(* IEC 61131-3 sources: Mizera_Tube/Plc (part 6) *)

(* ---- usrLoad.plc ---- *)
#funcdec "FLP.plc"
#funcdec "SPist.plc"

#include "usrMem.inc"
#include "Iol.inc"

VAR_IN_OUT
#include "usrIol.inc"
#include "mem.inc"
END_VAR

VAR
M1_M2_M3_MOVE:        SINGLE_PISTON;
CenteringPist1:       SINGLE_PISTON;
CenteringPist2:       SINGLE_PISTON;
CenteringPist3:       SINGLE_PISTON;
CenteringPist4:       SINGLE_PISTON;
Sup_G_Pist:           SINGLE_PISTON;
Pist_F_FB:            SINGLE_PISTON;
J_VEL_SWITCH:                    FF;
TON_CHAIN:                      TON;
TON_INVERTER_FIL:               TON;
TON_INVERTER_FIL1:              TON;
END_VAR

FUNCTION LOADER
************************************************************
* Loader Initialization Selection
************************************************************
PAGE_PLC

************************************************************
* Loader arms to be back (Arms J)
************************************************************
LD     ch0_ValFunM
EQ     330
OR(
LD     ch8_ValFunM
EQ     330
)
OR(
LD     ch0_ValFunM                * Arms J Going Back Slow
EQ     431
)
OR(
LD     ch0_ValFunM                * whole loader homming
EQ     445
)
AND    PRGRUN_CN0
ANDN   PRGSTOP_CN0
OR(
LD     BtnGuiM1M2M3_Open
ANDN   PRGRUN_CN0
)
ANDN   I_I_M1_M2_M3_OPEN
ST     O_O_M1_M2_M3_Open

LDN    I_I_M1_M2_M3_OPEN
AND(
LD     %ax30.ra92
LT     SUPPORT_4_Quota
)
ANDN   %cn0.rc8.0
ANDN   ch0_in_ref
S      %PLCmsg8.5

************************************************************
* Loader arms to be in machine (Arms J)
************************************************************
LD     ch0_ValFunM
EQ     331
OR(
LD     ch8_ValFunM
EQ     331
)
AND    PRGRUN_CN0
ANDN   PRGSTOP_CN0
OR(
LD     BtnGuiM1M2M3_Close
ANDN   PRGRUN_CN0
)
ANDN   I_I_M1_M2_M3_CLOSE
ST     O_O_M1_M2_M3_Close

CAL    TON_INVERTER_FIL(IN=I_I_M1_M2_M3_ALARM, PT=300)
LD     TON_INVERTER_FIL.Q
S      %PLCerr21.8

************************************************************
* Loader arms speed control
************************************************************
LD     O_O_M1_M2_M3_Close
OR(
       LD     ch0_ValFunM
       EQ     431                 * Slow Chain Backward
       AND    O_O_M1_M2_M3_Open
)
ANDN(
       LD     ch0_ValFunM
       EQ     330
       OR(
       LD     ch8_ValFunM
       EQ     330
       )
	   OR(
       LD     ch0_ValFunM                * whole loader homming
       EQ     445
       )
)
ORN    %cn0.rc8.0
ST     O_O_Arm_Slow

LDN    O_O_Arm_Slow
ST     O_O_Arm_Fast

************************************************************
* Loader chain to be inside (D)
************************************************************
LD     ch0_ValFunM
EQ     443
OR(
LD     ch8_ValFunM
EQ     443
)
AND    PRGRUN_CN0
ANDN   PRGSTOP_CN0
OR(
LD     BtnGuiChainForw
ANDN   I_I_TubeOnChain_D
ANDN   PRGRUN_CN0
)
ST     O_O_Chain_Forw_D

CAL    TON_CHAIN(IN=O_O_Chain_Forw_D,PT=20000) *20S
LD     TON_CHAIN.Q
AND    PRGRUN_CN0
S      STORE_Empty

CAL    TON_INVERTER_FIL1(IN=I_I_Loader_Alarm, PT=300)
LD     TON_INVERTER_FIL1.Q
S      %PLCerr21.9

************************************************************
* Loader chain to be outside (D)
************************************************************
LD     ch0_ValFunM
EQ     444
OR(
LD     ch8_ValFunM
EQ     444
)
AND    PRGRUN_CN0
ANDN   PRGSTOP_CN0
ANDN   I_I_HomeChain_E
OR(
LD     BtnGuiChainBackw
ANDN   PRGRUN_CN0
)
ST     O_O_Chain_Back_D

************************************************************
* Centering Piston 1
************************************************************
LD     PRGRUN_CN0                     ** M0.0 cn0.rc8.0  Programma in corso
ST     CenteringPist1.xAuto

LD     Pul_Reset                      ** (gPlc0.3)Reset pushbutton
OR     Pul_Start                      ** (gPlc0.1)Start pushbutton
ST     CenteringPist1.xReset

LD     BtnGuiCentering_Open_1
OR     BtnGuiCentering_Open_All
OR     Force_Open_Center_1
ST     CenteringPist1.xManualPlus

LD     BtnGuiCentering_Close_1
OR     BtnGuiCentering_Cls_All
ANDN   Force_Open_Center_1
ST     CenteringPist1.xManualMinus

LD     Fun_M332_Ch0
OR(
LD     ch8_ValFunM
EQ     332
)
OR     Fun_M445_Ch0
OR     Force_Open_Center_1
OR     Fun_M452_Ch0                   ** Open all centering
ST     CenteringPist1.xAutoPlus

LD     Fun_M333_Ch0
OR(
LD     ch8_ValFunM
EQ     333
)
OR     Fun_M455_Ch0
ST     CenteringPist1.xAutoMinus

LD     I_I_PRESSIONE_ARIA_IMPIANTO    ** **(Common for all pistons) %USR_M0
ST     CenteringPist1.xAirPressure

LD     I_I_Centering_Open_1
ST     CenteringPist1.xSensorPlus

LD     %PLCFLAGS.1
ST     CenteringPist1.xSensorMinus

LD     %PLCFLAGS.1
ST     CenteringPist1.xPlusAtInit

LD     %PLCFLAGS.1
ST     CenteringPist1.xSingleEffect

LD     10000
ST     CenteringPist1.xTimeOut

LDN    I_I_EMERGENZA                  ** Machine OK (no EMERG.)
ST     CenteringPist1.xEmerg

CAL    CenteringPist1

LD     CenteringPist1.yPistonPlus
ST     O_O_Centering_Open_1

LD     CenteringPist1.yPistonMinus
ST     O_O_Centering_Close_1

LD     CenteringPist1.yAlarm
ST     %PLCerr21.10

************************************************************
* Centering Piston 2
************************************************************
LD     PRGRUN_CN0                     ** M0.0 cn0.rc8.0  Programma in corso
ST     CenteringPist2.xAuto

LD     Pul_Reset                      ** (gPlc0.3)Reset pushbutton
OR     Pul_Start                      ** (gPlc0.1)Start pushbutton
ST     CenteringPist2.xReset

LD     BtnGuiCentering_Open_2
OR     BtnGuiCentering_Open_All
OR     Force_Open_Center_2
ST     CenteringPist2.xManualPlus

LD     BtnGuiCentering_Close_2
OR     BtnGuiCentering_Cls_All
ANDN   Force_Open_Center_2
ST     CenteringPist2.xManualMinus

LD     Fun_M446_Ch0
OR(
LD     ch8_ValFunM
EQ     446
)
OR     Fun_M445_Ch0
OR     Force_Open_Center_2
OR     Fun_M452_Ch0                   ** Open all centering
ST     CenteringPist2.xAutoPlus

LD     Fun_M447_Ch0
OR(
LD     ch8_ValFunM
EQ     447
)
OR     Fun_M455_Ch0
ST     CenteringPist2.xAutoMinus

LD     I_I_PRESSIONE_ARIA_IMPIANTO    ** **(Common for all pistons) %USR_M0
ST     CenteringPist2.xAirPressure

LD     I_I_Centering_Open_2
ST     CenteringPist2.xSensorPlus

LD     %PLCFLAGS.1
ST     CenteringPist2.xSensorMinus

LD     %PLCFLAGS.1
ST     CenteringPist2.xPlusAtInit

LD     %PLCFLAGS.1
ST     CenteringPist2.xSingleEffect

LD     10000
ST     CenteringPist2.xTimeOut

LDN    I_I_EMERGENZA                  ** Machine OK (no EMERG.)
ST     CenteringPist2.xEmerg

CAL    CenteringPist2

LD     CenteringPist2.yPistonPlus
ST     O_O_Centering_Open_2

LD     CenteringPist2.yPistonMinus
ST     O_O_Centering_Close_2

LD     CenteringPist2.yAlarm
ST     %PLCerr21.11

************************************************************
* Centering Piston 3
************************************************************
LD     PRGRUN_CN0                     ** M0.0 cn0.rc8.0  Programma in corso
ST     CenteringPist3.xAuto

LD     Pul_Reset                      ** (gPlc0.3)Reset pushbutton
OR     Pul_Start                      ** (gPlc0.1)Start pushbutton
ST     CenteringPist3.xReset

LD     BtnGuiCentering_Open_3
OR     BtnGuiCentering_Open_All
OR     Force_Open_Center_3
ST     CenteringPist3.xManualPlus

LD     BtnGuiCentering_Close_3
OR     BtnGuiCentering_Cls_All
ANDN   Force_Open_Center_3
ST     CenteringPist3.xManualMinus

LD     Fun_M448_Ch0
OR(
LD     ch8_ValFunM
EQ     448
)
OR     Fun_M445_Ch0
OR     Force_Open_Center_3
OR     Fun_M452_Ch0                   ** Open all centering
ST     CenteringPist3.xAutoPlus

LD     Fun_M449_Ch0
OR(
LD     ch8_ValFunM
EQ     449
)
OR     Fun_M455_Ch0
ST     CenteringPist3.xAutoMinus

LD     I_I_PRESSIONE_ARIA_IMPIANTO    ** **(Common for all pistons) %USR_M0
ST     CenteringPist3.xAirPressure

LD     I_I_Centering_Open_3
ST     CenteringPist3.xSensorPlus

LD     %PLCFLAGS.1
ST     CenteringPist3.xSensorMinus

LD     %PLCFLAGS.1
ST     CenteringPist3.xPlusAtInit

LD     %PLCFLAGS.1
ST     CenteringPist3.xSingleEffect

LD     10000
ST     CenteringPist3.xTimeOut

LDN    I_I_EMERGENZA                  ** Machine OK (no EMERG.)
ST     CenteringPist3.xEmerg

CAL    CenteringPist3

LD     CenteringPist3.yPistonPlus
ST     O_O_Centering_Open_3

LD     CenteringPist3.yPistonMinus
ST     O_O_Centering_Close_3

LD     CenteringPist3.yAlarm
ST     %PLCerr21.12

************************************************************
* Centering Piston 4
************************************************************
LD     PRGRUN_CN0                     ** M0.0 cn0.rc8.0  Programma in corso
ST     CenteringPist4.xAuto

LD     Pul_Reset                      ** (gPlc0.3)Reset pushbutton
OR     Pul_Start                      ** (gPlc0.1)Start pushbutton
ST     CenteringPist4.xReset

LD     BtnGuiCentering_Open_4
OR     BtnGuiCentering_Open_All
OR     Force_Open_Center_4
ST     CenteringPist4.xManualPlus

LD     BtnGuiCentering_Close_4
OR     BtnGuiCentering_Cls_All
ANDN   Force_Open_Center_4
ST     CenteringPist4.xManualMinus

LD     Fun_M450_Ch0
OR(
LD     ch8_ValFunM
EQ     450
)
OR     Fun_M445_Ch0
OR     Force_Open_Center_4
OR     Fun_M452_Ch0                   ** Open all centering
ST     CenteringPist4.xAutoPlus

LD     Fun_M451_Ch0
OR(
LD     ch8_ValFunM
EQ     451
)
OR     Fun_M455_Ch0
ST     CenteringPist4.xAutoMinus

LD     I_I_PRESSIONE_ARIA_IMPIANTO    ** **(Common for all pistons) %USR_M0
ST     CenteringPist4.xAirPressure

LD     I_I_Centering_Open_4
ST     CenteringPist4.xSensorPlus

LD     %PLCFLAGS.1
ST     CenteringPist4.xSensorMinus

LD     %PLCFLAGS.1
ST     CenteringPist4.xPlusAtInit

LD     %PLCFLAGS.1
ST     CenteringPist4.xSingleEffect

LD     10000
ST     CenteringPist4.xTimeOut

LDN    I_I_EMERGENZA                  ** Machine OK (no EMERG.)
ST     CenteringPist4.xEmerg

CAL    CenteringPist4

LD     CenteringPist4.yPistonPlus
ST     O_O_Centering_Open_4

LD     CenteringPist4.yPistonMinus
ST     O_O_Centering_Close_4

LD     CenteringPist4.yAlarm
ST     %PLCerr21.13

************************************************************
* Support ( G up / down )
************************************************************
LD     PRGRUN_CN0                     ** M0.0 cn0.rc8.0  Programma in corso
ST     Sup_G_Pist.xAuto

LD     Pul_Reset                      ** (gPlc0.3)Reset pushbutton
OR     Pul_Start                      ** (gPlc0.1)Start pushbutton
ST     Sup_G_Pist.xReset

LD     BtnGui_G_Up
ST     Sup_G_Pist.xManualPlus

LD     BtnGui_G_Dwn
ST     Sup_G_Pist.xManualMinus

LD     Fun_M334_Ch0
OR(
LD     ch8_ValFunM
EQ     334
)
ST     Sup_G_Pist.xAutoPlus          * Up

LD     Fun_M335_Ch0
OR(
LD     ch8_ValFunM
EQ     335
)
OR     Fun_M445_Ch0
ST     Sup_G_Pist.xAutoMinus         * Dwn

LD     I_I_PRESSIONE_ARIA_IMPIANTO    ** **(Common for all pistons) %USR_M0
ST     Sup_G_Pist.xAirPressure

LD     I_I_CylinderUp_G
ST     Sup_G_Pist.xSensorPlus

LD     I_I_CylinderDwn_G
ST     Sup_G_Pist.xSensorMinus

LD     %PLCFLAGS.0
ST     Sup_G_Pist.xPlusAtInit

LD     %PLCFLAGS.1
ST     Sup_G_Pist.xSingleEffect

LD     10000
ST     Sup_G_Pist.xTimeOut

LDN    I_I_EMERGENZA                  ** Machine OK (no EMERG.)
ST     Sup_G_Pist.xEmerg

CAL    Sup_G_Pist

LD     Sup_G_Pist.yPistonPlus
*ANDN   I_I_CylinderUp_G
ST     O_O_CylinderUp_G

LD     Sup_G_Pist.yPistonMinus
*ANDN   I_I_CylinderDwn_G
ST     O_O_CylinderDwn_G

LD     Sup_G_Pist.yAlarm
ST     %PLCerr20.13

************************************************************
* Support F (Forward/Backward)
************************************************************
LD     PRGRUN_CN0                     ** M0.0 cn0.rc8.0  Programma in corso
ST     Pist_F_FB.xAuto

LD     Pul_Reset                      ** (gPlc0.3)Reset pushbutton
OR     Pul_Start                      ** (gPlc0.1)Start pushbutton
ST     Pist_F_FB.xReset

LD     BtnGui_F_Forw
ST     Pist_F_FB.xManualPlus

LD     BtnGui_F_Backw
ST     Pist_F_FB.xManualMinus

LD     Fun_M434_Ch0
OR(
LD     ch8_ValFunM
EQ     434
)
ST     Pist_F_FB.xAutoPlus

LD     Fun_M435_Ch0
OR(
LD     ch8_ValFunM
EQ     435
)
OR(
LD     ch0_ValFunM                    * whole loader homming
EQ     445
)
ST     Pist_F_FB.xAutoMinus

LD     I_I_PRESSIONE_ARIA_IMPIANTO    ** **(Common for all pistons) %USR_M0
ST     Pist_F_FB.xAirPressure

LD     I_I_CylinderForw_F
ST     Pist_F_FB.xSensorPlus

LD     I_I_CylinderBack_F
ST     Pist_F_FB.xSensorMinus

LD     %PLCFLAGS.1
ST     Pist_F_FB.xPlusAtInit

LD     %PLCFLAGS.1
ST     Pist_F_FB.xSingleEffect

LD     10000
ST     Pist_F_FB.xTimeOut

LDN    I_I_EMERGENZA                  ** Machine OK (no EMERG.)
ST     Pist_F_FB.xEmerg

CAL    Pist_F_FB

LD     Pist_F_FB.yPistonPlus
ANDN   I_I_CylinderForw_F
ST     O_O_CylinderForw_F

LD     Pist_F_FB.yPistonMinus
ANDN   I_I_CylinderBack_F
ST     O_O_CylinderBack_F

LD     Pist_F_FB.yAlarm
ST     %PLCerr20.14

************************************************************
* Alarm / Status Reset
************************************************************
LD     Pul_Reset
ST     O_O_Rst_InverterAlm
R      %PLCmsg8.5
R      %PLCerr21.8
R      %PLCerr21.9
R      ISO_Loader_Retrace
R      iso_G510_Running
R      iso_G520_V_Unload
R      iso_G580_Running

LD     Pul_Reset
ORN    PRGRUN_CN0
R      STORE_Empty
R      TubeOnGworklist

LD     BtnClrLoaderBreakPoint
ANDN   %cn0.rc8.0
JMPCN  CLRLDSTATUS
LD     0
ST     LoaderProcess
CLRLDSTATUS:

END_FUNCTION

(* ---- usrMdec.plc ---- *)
**************************************************
********* READ M FROM ISO ************************
**************************************************
#defcom %rc9 Register M function
#defcom %rc8.4 Strobe M function

#include "usrMem.inc"

VAR_IN_OUT
#include "mem.inc"
END_VAR

VAR
Register_M_Ch0	             AT %cn0.rc9;
Strobe_M_Ch0  	             AT %cn0.rc8.4;
Register_M_Ch1	             AT %cn1.rc9;
Strobe_M_Ch1  	             AT %cn1.rc8.4;
Register_M_Ch2	             AT %cn2.rc9;
Strobe_M_Ch2  	             AT %cn2.rc8.4;
Register_M_Ch3	             AT %cn3.rc9;
Strobe_M_Ch3  	             AT %cn3.rc8.4;
Register_M_Ch4	             AT %cn4.rc9;
Strobe_M_Ch4  	             AT %cn4.rc8.4;
Register_M_Ch5	             AT %cn5.rc9;
Strobe_M_Ch5  	             AT %cn5.rc8.4;
Register_M_Ch7	             AT %cn7.rc9;
Strobe_M_Ch7  	             AT %cn7.rc8.4;
Register_M_Ch8	             AT %cn8.rc9;
Strobe_M_Ch8  	             AT %cn8.rc8.4;
END_VAR

FUNCTION USR_READ_M

* cn0

LD   Register_M_Ch0
EQ   330
AND  Strobe_M_Ch0
ST   Fun_M330_Ch0        * Open M1 M2 M3

LD   Register_M_Ch0
EQ   331
AND  Strobe_M_Ch0
ST   Fun_M331_Ch0        * Close M1 M2 M3

LD   Register_M_Ch0
EQ   332
AND  Strobe_M_Ch0
ST   Fun_M332_Ch0        * Open Centering Clamp

LD   Register_M_Ch0
EQ   333
AND  Strobe_M_Ch0
ST   Fun_M333_Ch0        * Close Centering Clamp

LD   Register_M_Ch0
EQ   334
AND  Strobe_M_Ch0
ST   Fun_M334_Ch0

LD   Register_M_Ch0
EQ   335
AND  Strobe_M_Ch0
ST   Fun_M335_Ch0

LD   Register_M_Ch0
EQ   336
AND  Strobe_M_Ch0
ST   Fun_M336_Ch0

LD   Register_M_Ch0
EQ   337
AND  Strobe_M_Ch0
ST   Fun_M337_Ch0

LD   Register_M_Ch0
EQ   338
AND  Strobe_M_Ch0
ST   Fun_M338_Ch0

LD   Register_M_Ch0
EQ   339
AND  Strobe_M_Ch0
ST   Fun_M339_Ch0

LD   Register_M_Ch0
EQ   431
AND  Strobe_M_Ch0
ST   Fun_M431_Ch0

LD   Register_M_Ch0
EQ   432
AND  Strobe_M_Ch0
ST   Fun_M432_Ch0

LD   Register_M_Ch0
EQ   434
AND  Strobe_M_Ch0
ST   Fun_M434_Ch0

LD   Register_M_Ch0
EQ   435
AND  Strobe_M_Ch0
ST   Fun_M435_Ch0

***
* M for Overlapped movement of the spindles

LD   Register_M_Ch0
EQ   440
AND  Strobe_M_Ch0
ST   Fun_M440_Ch0        * Move axis 30

LD   Register_M_Ch0
EQ   441
AND  Strobe_M_Ch0
ST   Fun_M441_Ch0        * Move axis 31

LD   Register_M_Ch0
EQ   442
AND  Strobe_M_Ch0
ST   Fun_M442_Ch0        * Move axis 36

LD   Register_M_Ch0
EQ   443
AND  Strobe_M_Ch0
ST   Fun_M443_Ch0

LD   Register_M_Ch0
EQ   444
AND  Strobe_M_Ch0
ST   Fun_M444_Ch0

LD   Register_M_Ch0
EQ   445
AND  Strobe_M_Ch0
ST   Fun_M445_Ch0

LD   Register_M_Ch0
EQ   446
AND  Strobe_M_Ch0
ST   Fun_M446_Ch0

LD   Register_M_Ch0
EQ   447
AND  Strobe_M_Ch0
ST   Fun_M447_Ch0

LD   Register_M_Ch0
EQ   448
AND  Strobe_M_Ch0
ST   Fun_M448_Ch0

LD   Register_M_Ch0
EQ   449
AND  Strobe_M_Ch0
ST   Fun_M449_Ch0

LD   Register_M_Ch0
EQ   450
AND  Strobe_M_Ch0
ST   Fun_M450_Ch0

LD   Register_M_Ch0
EQ   451
AND  Strobe_M_Ch0
ST   Fun_M451_Ch0

LD   Register_M_Ch0
EQ   452
AND  Strobe_M_Ch0
ST   Fun_M452_Ch0

LD   Register_M_Ch0
EQ   453
AND  Strobe_M_Ch0
ST   Fun_M453_Ch0

LD   Register_M_Ch0
EQ   454
AND  Strobe_M_Ch0
ST   Fun_M454_Ch0

LD   Register_M_Ch0
EQ   455
AND  Strobe_M_Ch0
ST   Fun_M455_Ch0

**

LD   Register_M_Ch0
EQ   720
AND  Strobe_M_Ch0
ST   Fun_M720_Ch0             ** Mobile spindle open

LD   Register_M_Ch0
EQ   721
AND  Strobe_M_Ch0
ST   Fun_M721_Ch0             ** Mobile spindle close

LD   Register_M_Ch0
EQ   722
AND  Strobe_M_Ch0
ST   Fun_M722_Ch0             ** Second mobile spindle open

LD   Register_M_Ch0
EQ   723
AND  Strobe_M_Ch0
ST   Fun_M723_Ch0             ** Second mobile spindle close

LD   Register_M_Ch0
EQ   724
AND  Strobe_M_Ch0
ST   Fun_M724_Ch0             ** Auto Up command for supports

LD   Register_M_Ch0
EQ   725
AND  Strobe_M_Ch0
ST   Fun_M725_Ch0             ** Auto Down Command

LD   Register_M_Ch0
EQ   726
AND  Strobe_M_Ch0
ST   Fun_M726_Ch0             ** Auto Up Command (Motor Following Support)

LD   Register_M_Ch0
EQ   730
AND  Strobe_M_Ch0
ST   Fun_M730_Ch0             * Request for load pipe

LD   Register_M_Ch0
EQ   731
AND  Strobe_M_Ch0
ST   Fun_M731_Ch0             * Request back loader

LD   Register_M_Ch0
EQ   732
AND  Strobe_M_Ch0
ST   Fun_M732_Ch0             * Read tube length

LD   Register_M_Ch0
EQ   733
AND  Strobe_M_Ch0
ST   Fun_M733_Ch0             * UP SUPP 1

LD   Register_M_Ch0
EQ   734
AND  Strobe_M_Ch0
ST   Fun_M734_Ch0             * UP SUPP 2

LD   Register_M_Ch0
EQ   735
AND  Strobe_M_Ch0
ST   Fun_M735_Ch0             * UP SUPP 3

LD   Register_M_Ch0
EQ   736
AND  Strobe_M_Ch0
ST   Fun_M736_Ch0             * UP SUPP 4

LD   Register_M_Ch0
EQ   825
AND  Strobe_M_Ch0
ST   Fun_M825_Ch0

LD   Register_M_Ch0
EQ   826
AND  Strobe_M_Ch0
ST   Fun_M826_Ch0

LD   Register_M_Ch0
EQ   827
AND  Strobe_M_Ch0
ST   Fun_M827_Ch0

LD   Register_M_Ch0
EQ   829
AND  Strobe_M_Ch0
ST   Fun_M829_Ch0

LD   Register_M_Ch0
EQ   830
AND  Strobe_M_Ch0
ST   Fun_M830_Ch0

LD   Register_M_Ch0
EQ   981
AND  Strobe_M_Ch0
ST   Fun_M981_Ch0

LD   Register_M_Ch0
EQ   982
AND  Strobe_M_Ch0
ST   Fun_M982_Ch0

LD   Register_M_Ch0
EQ   983
AND  Strobe_M_Ch0
ST   Fun_M983_Ch0

LD   Register_M_Ch0
EQ   984
AND  Strobe_M_Ch0
ST   Fun_M984_Ch0

LD   Register_M_Ch0
EQ   985
AND  Strobe_M_Ch0
ST   Fun_M985_Ch0

LD   Register_M_Ch0
EQ   986
AND  Strobe_M_Ch0
ST   Fun_M986_Ch0

LD   Register_M_Ch0
EQ   987
AND  Strobe_M_Ch0
ST   Fun_M987_Ch0

LD   Register_M_Ch0
EQ   988
AND  Strobe_M_Ch0
ST   Fun_M988_Ch0

LD   Register_M_Ch0
EQ   989
AND  Strobe_M_Ch0
ST   Fun_M989_Ch0

LD   Register_M_Ch0
EQ   990
AND  Strobe_M_Ch0
ST   Fun_M990_Ch0

LD   Register_M_Ch0
EQ   991
AND  Strobe_M_Ch0
ST   Fun_M991_Ch0

LD   Register_M_Ch0
EQ   992
AND  Strobe_M_Ch0
ST   Fun_M992_Ch0

LD   Register_M_Ch0
EQ   993
AND  Strobe_M_Ch0
ST   Fun_M993_Ch0

LD   Register_M_Ch0
EQ   994
AND  Strobe_M_Ch0
ST   Fun_M994_Ch0

END_FUNCTION

(* ---- UsrPLC.plc ---- *)
*******************************************************************************
*   MANAGEMENT USER PLC
*******************************************************************************

FUNCTION USR_INIT

#ifndef SIM_IO
USR_INP_CONFIG
#endif

SHARED_MEMORY

USR_READ_M

SPINDLES

LOADER

COMMAND_TO_MAIN

LOAD_SUPPORTS

LATERAL_SUPP

HORIZ_SUPP

UNLOAD_SUPPORTS

Lubrication

UNLOADER

*USR_MANAGEMENTS

M_WAIT

END_FUNCTION

FUNCTION USR_END

#ifndef SIM_IO
USR_OUT_CONFIG
#endif

END_FUNCTION

(* ---- usrPrntr.plc ---- *)
#include "usrMem.inc"

VAR
TON_Printer_Down:   TON;
TON_Printer_Up:     TON;
RT_Printer_Start:   R_TRIG;
END_VAR

VAR_IN_OUT

END_VAR

FUNCTION PRINTER

* CAL TON_Printer_Down(IN=O_O_Printer_Down,PT=2000)     * 2 sec
* CAL TON_Printer_Up(IN=O_O_Printer_Up,PT=2000)     * 2 sec
CAL RT_Printer_Start(CLK:=Fun_M342_Ch0)

* LD TON_Printer_Down.Q
LD I_I_Printer_Down
R  O_O_Printer_Down

LD Fun_M340_Ch0
S  O_O_Printer_Down

* LD TON_Printer_Up.Q
LD I_I_Printer_Up
R  O_O_Printer_Up

LD Fun_M341_Ch0
S  O_O_Printer_Up

LD RT_Printer_Start.Q
ST O_O_Printer_Start

END_FUNCTION

(* ---- usrSpind.plc ---- *)
#funcdec "assi.plc"
#funcdec "canfb.plc"
#funcdec "DynMng.plc"
#funcdec "FBSpindl.plc"
#funcdec "SPist.plc"
#funcdec "cnc.plc"
#funcdec "Antictrl.plc"

#include "usrMem.inc"
#include "Iol.inc"

VAR
#include "cnc.inc"
MainSpindle:           SINGLE_PISTON;
SlaveSpindle:          SPINDLE;
MidSpindle:            SPINDLE;

MobSpZDiam:            LINEAR_CALC;
MobSpYDiam:            LINEAR_CALC;

FixSpZDiam:            LINEAR_CALC;
FixSpYDiam:            LINEAR_CALC;

TOF_Close_Spindle:     TOF;
TOF_Open_Spindle:      TOF;
R_TRIG_INIT:           R_TRIG;
R_TRIG_POSSIBLE_COL:   R_TRIG;

appoggio:              BOOL;
OPEN_SPIN_IN_AUTO:     BOOL;
DistU:                 DWORD;
DistV:                 DWORD;
SafeDistAppoggio:      DWORD;

DistX:                 DWORD;
DistY:                 DWORD;

AncolliXW:             ANTI_AXIS;
AncolliWV:             ANTI_AXIS;
POS_AX30:              AX_POSIZ;
POS_AX31:              AX_POSIZ;

MoveAx30_Jog:           BOOL;
PosToReachAx30:        DWORD;

MoveAx31_Jog:           BOOL;
PosToReachAx31:        DWORD;
END_VAR

VAR_IN_OUT
#include "mem.inc"
#include "usrIol.inc"
END_VAR

FUNCTION SPINDLES

**********************************************************************
* First Mobile Spindle
**********************************************************************
LD   PRGRUN_CN0                     ** M0.0 cn0.rc8.0  Programma in corso
ST   MainSpindle.xAuto

LD   Pul_Reset                      ** (gPlc0.3)Reset pushbutton
OR   Pul_Start                      ** (gPlc0.1)Start pushbutton
ST   MainSpindle.xReset

LD   MS_Open_Button
OR   I_I_Pul_Mobile_Spindle_Open
ST   MainSpindle.xManualPlus

LD   MS_Close_Button
OR   I_I_Pul_Mobile_Spindle_Close
ST   MainSpindle.xManualMinus

LD   Fun_M720_Ch0
ST   MainSpindle.xAutoPlus

LD   Fun_M721_Ch0
ST   MainSpindle.xAutoMinus

LD   I_I_PRESSIONE_ARIA_IMPIANTO
ST   MainSpindle.xAirPressure

*LD   I_I_Mobile_Spindle_Open
LD   O_O_Mobile_Spindle_Open
ST   MainSpindle.xSensorPlus

*LD   I_I_Mobile_Spindle_Close
LD   O_O_Mobile_Spindle_Close
ST   MainSpindle.xSensorMinus

LD   MainSpdLastOpen
ST   MainSpindle.xPlusAtInit

LD   %PLCFLAGS.0
ST   MainSpindle.xSingleEffect

LD   Time_Out_Sp
ST   MainSpindle.xTimeOut

LDN  I_I_EMERGENZA                  ** Machine OK (no EMERG.)
ST   MainSpindle.xEmerg

CAL  MainSpindle

LD   MainSpindle.yPistonPlus
ST   O_O_Mobile_Spindle_Open
ST   TM32_Mobile_Spindle_Open
S    MainSpdLastOpen

LD   MainSpindle.yPistonMinus
ST   O_O_Mobile_Spindle_Close
R    MainSpdLastOpen

********************************************************************************
* Middle Spindle Management (W)
********************************************************************************
*LD   I_I_FixedSpindle_Open
LD   O_O_SpindleFix_Open
OR(
LD   %PLCFLAGS.8
AND  MidSpdLastOpen
)
ST   MidSpindle.xSpOpen

*LD   I_I_FixedSpindle_Close
LD   O_O_SpindleFix_Close
ST   MidSpindle.xSpClose

LD   I_I_EMERGENZA
OR   EMER_GEN
ST   MidSpindle.xEmerg

LD   ProgRunCh0
ST   MidSpindle.xProgRun

LD   Fun_M982_Ch0
ST   MidSpindle.xAutoClose

LD   Fun_M981_Ch0
ST   MidSpindle.xAutoOpen

LD   FixedSpindleClose_Button
ST   MidSpindle.xManualClose

LD   FixedSpindleOpen_Button
ST   MidSpindle.xManualOpen

LD   Time_Out_Sp
ST   MidSpindle.xTimeout

LD   %TabLsr1.L_Tickness
ST   MidSpindle.xThickness

LD   ResAnalogPressure
ST   MidSpindle.xResOut

LD   120
ST   MidSpindle.xIndGraphPress

LD   I_I_Pressure_Mobile
ST   MidSpindle.xFeedbkPress

CAL  MidSpindle

LD   MidSpindle.yOpen
ST   O_O_SpindleFix_Open
ST   TM32_SpindleFix_Open
S    MidSpdLastOpen

LD   MidSpindle.yClose
ST   O_O_SpindleFix_Close
R    MidSpdLastOpen

**********************************************************************
* Second Mobile Spindle (V)
**********************************************************************
LD   I_I_EMERGENZA
OR   EMER_GEN
ST   SlaveSpindle.xEmerg

*LD   I_I_Mobile_Spindle_Slave_Open
LD   O_O_Mobile_Spindle_Slave_Open
OR(
LD   %PLCFLAGS.8
AND  SlaveSpdLastOpen
)
ST   SlaveSpindle.xSpOpen

*LD   I_I_Mobile_Spindle_Slave_Close
LD   O_O_Mobile_Spindle_Slave_Close
ST   SlaveSpindle.xSpClose

LD   ProgRunCh0
ST   SlaveSpindle.xProgRun

LD   Fun_M723_Ch0
ST   SlaveSpindle.xAutoClose

LD   Fun_M722_Ch0
ST   SlaveSpindle.xAutoOpen

LD   SMobile_Close_Button
ST   SlaveSpindle.xManualClose

LD   SMobile_Open_Button
ST   SlaveSpindle.xManualOpen

LD   Time_Out_Sp
ST   SlaveSpindle.xTimeout

LD   %TabLsr1.L_Tickness
ST   SlaveSpindle.xThickness

LD   ResAnalogPressure
ST   SlaveSpindle.xResOut

LD   121
ST   SlaveSpindle.xIndGraphPress

LD   I_I_Pressure_Fix
ST   SlaveSpindle.xFeedbkPress

CAL  SlaveSpindle

LD   SlaveSpindle.yBrake
ST   O_O_Mobile_Spindle_Slave_Brake

LD   SlaveSpindle.yOpen
ORN  %cn3.cc1.4                       *Exsisting V axis
ST   O_O_Mobile_Spindle_Slave_Open
ST   TM32_Mobile_Spindle_Slave_Open
S    SlaveSpdLastOpen

LD   SlaveSpindle.yClose
AND  %cn3.cc1.4                       *Exsisting V axis
ST   O_O_Mobile_Spindle_Slave_Close
R    SlaveSpdLastOpen

LD   SlaveSpindle.yAnOutPress
ST   O_O_Pressure_MobileS

LD   SlaveSpindle.yOutPressBar
ST   MobileSClosePressReq

LD   SlaveSpindle.yActualPressFeedbk
ST   PressMobileSClose

*******************************************************************************
* C1 and head emer safety
*******************************************************************************
LDN  Gest5Ax
AND  %cn3.cc1.5
JMPCN SKIPNON5AX

LD   %ax29.pa22
SUB  %ax29.ra4
ABS
GT   20000
OR   (
LD   %ax28.pa21
SUB  %ax28.ra4
ABS
GT   20000
)
ST   Hold_moving_axW

LD   %ax29.ra0.9   * Z-
OR   %ax28.ra0.8   * Y+
OR   %ax36.ra0.9   * W-
AND(
LD   %ax36.pa22
SUB  %ax36.ra4
GT   5000
)
AND(
LD   %ax36.ra4
GE   0
)
OR  (
     LD   %ax29.ra0.9  * Z-
     OR   %ax28.ra0.8  * Y+
     OR   %ax36.ra0.8  * W+
     AND(
     LD   %ax36.ra4
     SUB  %ax36.pa21
     GT   5000
     )
   	 AND(
     LD   %ax36.ra4
     LT   0
     )
)
AND  Hold_moving_axW
ANDN ch0_in_ref
ANDN %PlcOp0.22
S    %PLCerr20.22

SKIPNON5AX:

*******************************************************************************
* WV Emer safety
*******************************************************************************
LD   %ax36.ra4
SUB  %ax31.ra4
ABS
LT   Emer_SafeDis_WV *210000
OR	 (
LD   %ax36.ra4
SUB  %ax30.ra4
ABS
LT   Emer_SafeDis_XW *430000
)
ANDN ch0_in_ref
ST   appoggio

CAL  R_TRIG_POSSIBLE_COL(CLK=appoggio)
LD   R_TRIG_POSSIBLE_COL.Q
AND  %cn3.cc1.4
AND  %cn3.cc1.5
ANDN %PlcOp0.22
S    %PLCerr20.23

LD   Pul_Reset
R    %PLCerr20.22
R    %PLCerr20.23

*******************************************************************************
* XW Hold Safety
*******************************************************************************
LD   ECAT_OK
OR   MACC_TARATA
ST   appoggio
CAL  R_TRIG_INIT(CLK=appoggio)

LD   ALWAYS_ONE
ST   AncolliXW.xAx1_Fst

LD   Reset
OR   R_TRIG_INIT.Q
ST   AncolliXW.xReset

LD   36
ST   AncolliXW.xAx1_Num

LD   30
ST   AncolliXW.xAx2_Num

LD   SafeDis_XW
ST   AncolliXW.xDisSafe

CAL  AncolliXW

LD   AncolliXW.yHoldMov
AND  %cn3.cc1.5
ANDN %PlcOp0.22
ST   AncolliXW_yHoldMov
ST   %PLCerr20.20

*******************************************************************************
* WV Hold Safety
*******************************************************************************
LD   ALWAYS_ZERO
ST   AncolliWV.xAx1_Fst

LD   Reset
OR   R_TRIG_INIT.Q
ST   AncolliWV.xReset

LD   36
ST   AncolliWV.xAx1_Num

LD   31
ST   AncolliWV.xAx2_Num

LD   SafeDis_WV
ST   AncolliWV.xDisSafe

CAL  AncolliWV

LD   AncolliWV.yHoldMov
AND  %cn3.cc1.4
AND  %cn3.cc1.5
ANDN %PlcOp0.22
ST   AncolliWV_yHoldMov
ST   %PLCerr20.21

********************************************************************************
* Auto Spindle Movement

PATH %ax30

LD   Fun_M440_Ch0
AND  ProgRunCh0                     * program in run ch0
S    MoveAx30_Auto

LD   MoveAx30GuiBtn
AND  Ch0_Jog
S    MoveAx30_Jog

LD   MoveAx30_Jog
OR   MoveAx30_Auto
ST   POS_AX30.xax_ENABLE

LDN  POS_AX30.xax_ENABLE
ST   POS_AX30.xax_CLEAR

LD   POS_AX30.xax_ENABLE
AND  POS_AX30.yax_READY
ANDN POS_AX30.yax_ENDOK
ANDN POS_AX30.yax_ENDERR
ST   POS_AX30.xax_START

LD   PosSpindleX
ST   PosToReachAx30

LD   PosToReachAx30
GT   %pa22
OR   (
LD   PosToReachAx30
LT   %pa21
)
AND  Fun_M440_Ch0
S    %PLCmsg1.18        ** X axis positioning out of range

LD   Reset
R    %PLCmsg1.18

LD   PosToReachAx30
GT   %pa22
JMPCN no_pos_lim

LD   %pa22
ST   PosToReachAx30
no_pos_lim:

LD   PosToReachAx30
LT   %pa21
JMPCN no_neg_lim

LD   %pa21
ST   PosToReachAx30
no_neg_lim:

LD   PosToReachAx30
ST   POS_AX30.xax_QUOTA

LD   MoveAx30_Auto
JMPCN noVelAuto
LD   VelPosSpindleX_Auto
ST   POS_AX30.xax_VEL
JMP  noVelMan
noVelAuto:

LD   %pa9
DIV  3
ST   POS_AX30.xax_VEL
noVelMan:

CAL  POS_AX30

LD   POS_AX30.yax_ENDOK
AND  POS_AX30.xax_ENABLE
OR   Reset                            ** Reset Command
* OR   (
* LD   %ra4
* DIV  20
* EQ (
* LD   PosSpindleX
* DIV  20
* )
* )
R    MoveAx30_Auto                    ** (LsPlc63.0) Lens positioning finish
R    MoveAx30_Jog

LD   POS_AX30.xax_ENABLE
ST   GrantPlcMoveX

*

PATH %ax31

LD   Fun_M441_Ch0
AND  ProgRunCh0                     * program in run ch0
S    MoveAx31_Auto

LD   MoveAx31GuiBtn
AND  Ch0_Jog
S    MoveAx31_Jog

LD   MoveAx31_Jog
OR   MoveAx31_Auto
ST   POS_AX31.xax_ENABLE

LDN  POS_AX31.xax_ENABLE
ST   POS_AX31.xax_CLEAR

LD   POS_AX31.xax_ENABLE
AND  POS_AX31.yax_READY
ANDN POS_AX31.yax_ENDOK
ANDN POS_AX31.yax_ENDERR
ST   POS_AX31.xax_START

LD   PosSpindleX1
ST   PosToReachAx31

LD   PosToReachAx31
GT   %pa22
OR   (
LD   PosToReachAx31
LT   %pa21
)
AND  Fun_M441_Ch0
S    %PLCmsg1.17        ** V axis positioning out of range

LD   Reset
R    %PLCmsg1.17

LD   PosToReachAx31
GT   %pa22
JMPCN no_pos_lim1

LD   %pa22
ST   PosToReachAx31
no_pos_lim1:

LD   PosToReachAx31
LT   %pa21
JMPCN no_neg_lim1

LD   %pa21
ST   PosToReachAx31
no_neg_lim1:

LD   PosToReachAx31
ST   POS_AX31.xax_QUOTA

LD   MoveAx31_Auto
JMPCN noVelAuto1
LD   VelPosSpindleX1_Auto
ST   POS_AX31.xax_VEL
JMP  noVelMan1
noVelAuto1:

LD   %pa9
DIV  3
ST   POS_AX31.xax_VEL
noVelMan1:

CAL  POS_AX31

LD   POS_AX31.yax_ENDOK
AND  POS_AX31.xax_ENABLE
OR   Reset                            ** Reset Command
* OR   (
* LD   %ra4
* DIV  20
* EQ (
* LD   PosSpindleX1
* DIV  20
* )
* )
R    MoveAx31_Auto                    ** (LsPlc63.0) Lens positioning finish
R    MoveAx31_Jog

LD   POS_AX31.xax_ENABLE
ST   GrantPlcMoveX1

********************************************************************************

END_FUNCTION

(* ---- usrSuppo.plc ---- *)
#funcdec "FBSuppor.plc"
#funcdec "assi.plc"
#funcdec "DynMng.plc"
#funcdec "FBAux.plc"
#funcdec "SupForce.plc"
#funcdec "suppFB.plc"

#include "Iol.inc"
#include "usrMem.inc"

VAR
#include "iof.inc"
#include "usrIof.inc"
#include "cnc.inc"

F_TRIG_RES_FOLL:     F_TRIG;

appoggio:              BOOL;

SUP1:               SUPPORT;
SUP2:               SUPPORT;
SUP3:               SUPPORT;
SUP4:               SUPPORT;
END_VAR

VAR_IN_OUT
#include "usrIol.inc"
#include "mem.inc"
END_VAR

FUNCTION LOAD_SUPPORTS

PATH  %cn5

*******************************************************
*         Staggered avoidance position                *
*******************************************************
LD   %ax30.ra0.0
JMPCN _closeloop_active
     LD   %ax30.ra92
     ST   PosUMis
JMP _no_loop
_closeloop_active:
     LD   %ax30.ra4
     ST   PosUMis
_no_loop:

LDN  OptEnabAutoParkLoad
JMPCN _DISABLEFOLLOWER
     LD   0
     ST   PosUMis
_DISABLEFOLLOWER:

*******************************************************
*         FOLLOWIING SUPPORTS MANAGEMENT              *
*******************************************************
 *(gIso39.0) Enable blendSwitch PLC writes (Lunette da ISO)
CAL  F_TRIG_RES_FOLL (CLK:=PRGRUN_CN0)
LD   F_TRIG_RES_FOLL.Q
OR   Pul_Reset
R    EnWriteBlendSwitch1
R    ParkAllLoadSuppCmd

LDN  PRGRUN_CN0
JMPCN RSTBLEND
     LD   %PLCFLAGS.0
	 ST   EnWriteBlendSwitch1
	 ST   ISO_SupLoader_Init
	 ST   ParkUn51Sup_ISO
	 ST   ParkUn52Sup_ISO
	 ST   ParkUn53Sup_ISO
	 ST   ParkUn54Sup_ISO

     LD   0
	 ST   ThreshLoadingSupDown
RSTBLEND:

LD   ALWAYS_ONE
ST   SUP1.xUaxDir
ST   SUP2.xUaxDir
ST   SUP3.xUaxDir
ST   SUP4.xUaxDir

LD   Reset
OR   EMER_GEN
ST   SUP1.xReset
ST   SUP2.xReset
ST   SUP3.xReset
ST   SUP4.xReset

LD   EnWriteBlendSwitch1
ST   SUP1.xBlendSwitchEn
ST   SUP2.xBlendSwitchEn
ST   SUP3.xBlendSwitchEn
ST   SUP4.xBlendSwitchEn

LD   OptEnabAutoParkLoad
ST   SUP1.xEnabAutoDwn
ST   SUP2.xEnabAutoDwn
ST   SUP3.xEnabAutoDwn
ST   SUP4.xEnabAutoDwn

LD   IN_M700_M704
EQ   700
OR(
LD   IN_M700_M704
EQ   704
)
AND  %cn0.rc8.0
JMPC CLRACTBIT
     LD   %PLCFLAGS.0
     ST   M700_BLEND
CLRACTBIT:

LD   IN_M700_M704
EQ   704
OR   M700_BLEND
AND  %cn0.rc8.0
AND  O_O_Mobile_Spindle_Close
ANDN IN_M4_MODE
ST   SUP1.xEnabAutoUp
ST   SUP2.xEnabAutoUp
ST   SUP3.xEnabAutoUp
ST   SUP4.xEnabAutoUp

LD   IN_M700_M704
ST   SUP1.xM700_M704
ST   SUP2.xM700_M704
ST   SUP3.xM700_M704
ST   SUP4.xM700_M704

LD   IN_M4_MODE
JMPCN NOG1000PRK
     LD   0
     ST   SUP1.xM700_M704
     ST   SUP2.xM700_M704
     ST   SUP3.xM700_M704
     ST   SUP4.xM700_M704
NOG1000PRK:

LD   PosUMis
ST   SUP1.xSupervisePos
ST   SUP2.xSupervisePos
ST   SUP3.xSupervisePos
ST   SUP4.xSupervisePos

LD   ParkingPositionLoad
ST   SUP1.xParkingPos
ST   SUP2.xParkingPos
ST   SUP3.xParkingPos
ST   SUP4.xParkingPos

LD   ThreshLoadingSupDown
ST   SUP1.xSuperviseOft
ST   SUP2.xSuperviseOft
ST   SUP3.xSuperviseOft
ST   SUP4.xSuperviseOft

LD   %ax30.ra3.0
ST   SUP1.xUaxStill
ST   SUP2.xUaxStill
ST   SUP3.xUaxStill
ST   SUP4.xUaxStill

* [lv, lat, ulv, uhor]=[0,1,2,3]
LD   0
ST   SUP1.xBlendId
ST   SUP2.xBlendId
ST   SUP3.xBlendId
ST   SUP4.xBlendId

LD   %config_machine0.7
ST   SUP1.xEnCyComSup
ST   SUP2.xEnCyComSup
ST   SUP3.xEnCyComSup
ST   SUP4.xEnCyComSup
JMPCN _CYCOMOFT
LD   %ax60.ra24
ST   SUP1.xCyComOft
ST   SUP2.xCyComOft
ST   SUP3.xCyComOft
ST   SUP4.xCyComOft
_CYCOMOFT:

* Support 1
LD   %cn5.cc1.1
JMPCN no_support_1

PATH  %ax51

LD   SUPPORT_1_Quota
ST   SUP1.xLimitSuppDwn

LD   ParkAllLoadSuppCmd
OR   Fun_M725_Ch0
OR   ParkUn51Sup_ISO
ST   SUP1.xParkCmd

CAL  SUP1

LD   SUP1.yReqGrant
ANDN ch5_in_ref
ST   usrReqGrantSupL1

LD   SUP1.yHoldMovSupp
ANDN ch5_in_ref
ST   HoldZ1SuppLoad

LD   SUP1.yHoldMovSuperv
ANDN ch5_in_ref
ST   Hold_U_Z1SuppLoad

LD   SUP1.yCenterOpen
ST   Force_Open_Center_1

LD   SUP1.yCyComDwn
ST   yActivatedCyCom_51

LD   SUP1.yCyComOft
ST   CyComOftAx51

no_support_1:

* Support 2

LD   %cn5.cc1.2
JMPCN no_support_2

PATH  %ax52

LD   SUPPORT_2_Quota
ST   SUP2.xLimitSuppDwn

LD   ParkAllLoadSuppCmd
OR   Fun_M725_Ch0           * M force parking from autocycle
OR   ParkUn52Sup_ISO
ST   SUP2.xParkCmd

CAL  SUP2

LD   SUP2.yReqGrant
ANDN ch5_in_ref
ST   usrReqGrantSupL2

LD   SUP2.yHoldMovSupp
ANDN ch5_in_ref
ST   HoldZ2SuppLoad

LD   SUP2.yHoldMovSuperv
ANDN ch5_in_ref
ST   Hold_U_Z2SuppLoad

LD   SUP2.yCenterOpen
ST   Force_Open_Center_2

LD   SUP2.yCyComDwn
ST   yActivatedCyCom_52

LD   SUP2.yCyComOft
ST   CyComOftAx52

no_support_2:

*  Support 3
*
LD   %cn5.cc1.3
JMPCN no_support_3

PATH  %ax53

LD   SUPPORT_3_Quota            * dwn limit for support
ST   SUP3.xLimitSuppDwn

LD   ParkAllLoadSuppCmd
OR   Fun_M725_Ch0           * M force parking from autocycle
OR   ParkUn53Sup_ISO
ST   SUP3.xParkCmd

CAL  SUP3

LD   SUP3.yReqGrant
ANDN ch5_in_ref
ST   usrReqGrantSupL3

LD   SUP3.yHoldMovSupp
ANDN ch5_in_ref
ST   HoldZ3SuppLoad

LD   SUP3.yHoldMovSuperv
ANDN ch5_in_ref
ST   Hold_U_Z3SuppLoad

LD   SUP3.yCenterOpen
ST   Force_Open_Center_3

LD   SUP3.yCyComDwn
ST   yActivatedCyCom_53

LD   SUP3.yCyComOft
ST   CyComOftAx53

no_support_3:

*  Support 4
*
LD   %cn5.cc1.4
JMPCN no_support_4

PATH  %ax54

LD   SUPPORT_4_Quota            * dwn limit for support
ST   SUP4.xLimitSuppDwn

LD   ParkAllLoadSuppCmd
OR   Fun_M725_Ch0           * M force parking from autocycle
OR   ParkUn54Sup_ISO
ST   SUP4.xParkCmd

CAL  SUP4

LD   SUP4.yReqGrant
ANDN ch5_in_ref
ST   usrReqGrantSupL4

LD   SUP4.yHoldMovSupp
ANDN ch5_in_ref
ST   HoldZ4SuppLoad

LD   SUP4.yHoldMovSuperv
ANDN ch5_in_ref
ST   Hold_U_Z4SuppLoad

LD   SUP4.yCenterOpen
ST   Force_Open_Center_4

LD   SUP4.yCyComDwn
ST   yActivatedCyCom_54

LD   SUP4.yCyComOft
ST   CyComOftAx54

no_support_4:

*//=============================================================================
*// Cylinder Type Follower Support
*//=============================================================================
LOAD_CYLINDER_SUPPORTS

*//=============================================================================

END_FUNCTION

(* ---- usrSupUn.plc ---- *)
#funcdec "assi.plc"
#funcdec "suppFB.plc"
#funcdec "SPist.plc"
#funcdec "DynMng.plc"
#funcdec "FBAux.plc"
#funcdec "SupForce.plc"

#include "usrMem.inc"
#include "Iol.inc"

VAR
#include "iof.inc"
#include "usrIof.inc"
#include "cnc.inc"

appoggio:                      BOOL;
AllowSecFTar:                  BOOL;
M700_OR_M704:                  BOOL;
TubeReachSup_71:               BOOL;
TubeReachSup_72:               BOOL;
TubeReachSup_73:               BOOL;
TubeReachSup_74:               BOOL;
TubeReachSup_75:               BOOL;

TP_BIN_DOOR:                     TP;
RTRIG_RES_PRK:        	     R_TRIG;
R_Trig_UseCent:              R_TRIG;
RTRIG_Heading:               R_TRIG;
Rtrig_TubeInMac:             R_TRIG;
RTrig_SetFollow:             R_TRIG;
RTRIG_RES_GEA_OPT:           R_TRIG;
FTrig_SetFollow:             F_TRIG;
F_TRIG_RES_FOLL:             F_TRIG;

SUP71:                      SUPPORT;
SUP72:                      SUPPORT;
SUP73:                      SUPPORT;
SUP74:                      SUPPORT;
SUP75:                      SUPPORT;

CALQ_PRESTOP_V:        CALQ_PRESSLV;
SUP71_ForceDwn:  ISO_SUP_FORCE_DOWN;
SUP72_ForceDwn:  ISO_SUP_FORCE_DOWN;
SUP73_ForceDwn:  ISO_SUP_FORCE_DOWN;
SUP74_ForceDwn:  ISO_SUP_FORCE_DOWN;
SUP75_ForceDwn:  ISO_SUP_FORCE_DOWN;
END_VAR

VAR_IN_OUT
#include "usrIol.inc"
#include "mem.inc"
END_VAR

FUNCTION UNLOAD_SUPPORTS

PATH  %cn8

*******************************************************
* Unloading Vertical and Horizontal Sup VEL BLENDER
*******************************************************
*CALC_BLD_FEED
BLEND_FEEDRATE

*******************************************************
* Allow tube head avoidance
*******************************************************
LD   IN_M700_M704
EQ   700
OR(
LD   IN_M700_M704
EQ   704
)
AND  %cn0.rc8.0
ST   M700_OR_M704

LD   %cn0.rc8.0
AND  EnWriteBlendSwitch        * Unload
ANDN M700_OR_M704
ANDN Dis2ndFlapTar
ANDN %ax0.ra3.0
ANDN %ax0.ra3.2
ANDN IN_M4_MODE
ST   AllowSecFTar

*******************************************************
* Staggered avoidance position
*******************************************************
PATH %ax31
LD   IN_M4_MODE
OR   IN_M3_MODE
ANDN iso_G520_Running
AND  %cn0.rc8.0
ST   appoggio
CAL  CALQ_PRESTOP_V(xEn:=appoggio,xQta:=%ax31.ra92,xSpdNum:=3)
LD   CALQ_PRESTOP_V.Q
ST   SupervisePos_X1

LDN  %ax31.ra3.2    *Forward Movement of Slave Spindle
ANDN %ax31.ra3.0
JMPCN BCKWARDX1CASE
LD   %ax31.ra4
ST   SupervisePos_X1
BCKWARDX1CASE:

LDN  %cn3.cc1.4     *Exsisting V axis
JMPCN CASENO3SPINDLE
     LD   -9999999
     ST   SupervisePos_X1
CASENO3SPINDLE:

*******************************************************
* Tube Length In the machine
*******************************************************
LD   ResetTubeInMac
ANDN PRGRUN_CN0
ST   appoggio
CAL  Rtrig_TubeInMac(CLK:=appoggio)
LD   Rtrig_TubeInMac.Q
JMPCN no_tube
LD   %ax30.ra4
SUB (                                * In G800, should ensure always heading without angle
     LD  %ax33.ra4
     SIN
	 MULDIV(M=%twi1.htwi.oarh.dZ,D=1000)
)
ST   PosUHeading                     * last U heading position
no_tube:

CAL  RTRIG_Heading (CLK:=iso_pipeinside_mngt)
LD   RTRIG_Heading.Q
JMPCN  no_req_U_pos
LD   %ax30.ra4
ST   PosUHeading                     * last U heading position
no_req_U_pos:

LD   PosUHeading                     * Last U heading cut position
SUB  %ax30.ra4                       * U axis Position
* ADD is correct here, to avoid following support up/down during bevel cutting
ADD (                                * In G800, should ensure always heading without angle
     LD  %ax33.ra4
     SIN
	 MULDIV(M=%twi1.htwi.oarh.dZ,D=1000)
)
ST   TubeLengthInMach                * Tube present after the fixed spindle

LD   TubeLengthInMach
LT   0
JMPCN LengthNotDefined
LD   0
ST   TubeLengthInMach
LengthNotDefined:

LD   %ServiceMillePGM.13
JMPCN Not_manual_follow
LD   %ax30.pa22
ST   TubeLengthInMach
Not_manual_follow:

LD   O_O_SpindleFix_Close
AND  O_O_Mobile_Spindle_Slave_Close
ANDN O_O_Mobile_Spindle_Close
ST   IN_M4_MODE

LD   O_O_SpindleFix_Close
AND  O_O_Mobile_Spindle_Slave_Close
AND  O_O_Mobile_Spindle_Close
ST   IN_M3_MODE

LD   O_O_SpindleFix_Close
ANDN O_O_Mobile_Spindle_Slave_Close
AND  O_O_Mobile_Spindle_Close
ST   IN_M2_MODE

*******************************************************
* Dust Bin Management (1 == UP)
*******************************************************
LD   iso_bincmd
AND  PRGRUN_CN0
OR(
LD   gui_binup
ANDN PRGRUN_CN0
)
ANDN (
LD   %ax36.ra4
LT   SafeDis_W_Dustbin                * Less, not allow dustbin up
)
OR   O_O_Flap_Incline
OR(
LD   O_O_Flap_Home
ANDN I_I_Flap_Home
)
ST   O_O_Bin_Door     * (1 == UP)

LD   Pul_Reset
R    iso_bincmd
R    gui_binup

*******************************************************
*         FOLLOWIING SUPPORTS MANAGEMENT              *
*******************************************************
CAL  F_TRIG_RES_FOLL (CLK:=PRGRUN_CN0)
LD   F_TRIG_RES_FOLL.Q
OR   Pul_Reset
R    EnWriteBlendSwitch
R    CmdBlendSwitch
R    ParkAllCmd
R    AllFlapsHome
R    AllFlapsIncline

LD   iso_G520_Running
AND  %cn0.rc8.1
ST   HoldFlapInclined
R    AllFlapsHome
R    AllFlapsIncline
R    InclineFlapL1_ISO
R    InclineFlapL2_ISO
R    InclineFlapL3_ISO
R    InclineFlapL4_ISO
R    InclineFlapL5_ISO

LDN  PRGRUN_CN0
JMPCN RSTBLEND
     LD   %PLCFLAGS.0
     ST   EnWriteBlendSwitch
     ST   CmdBlendSwitch
     ST   ParkUn71Sup_ISO
	 ST   ParkUn72Sup_ISO
	 ST   ParkUn73Sup_ISO
	 ST   ParkUn74Sup_ISO
	 ST   ParkUn75Sup_ISO
	 ST   InclineFlapL1_ISO
	 ST   InclineFlapL2_ISO
	 ST   InclineFlapL3_ISO
	 ST   InclineFlapL4_ISO
	 ST   InclineFlapL5_ISO
	 ST   ISO_SupUn_Init
	 ST   ISO_Loader_Ack
	 ST   ISO_Loader_Req

	 LD   0
	 ST   OffsetUnSuppDwn_71
     ST   OffsetUnSuppDwn_72
	 ST   UpSupVoffset
	 ST   IN_M700_M704
RSTBLEND:

LD   Reset
OR   EMER_GEN
ST   SUP71.xReset
ST   SUP72.xReset
ST   SUP73.xReset
ST   SUP74.xReset
ST   SUP75.xReset

LD   ISO_SupUn_Init
ST   SUP71.xHoldExem
ST   SUP72.xHoldExem
ST   SUP73.xHoldExem
ST   SUP74.xHoldExem
ST   SUP75.xHoldExem

LD   EnWriteBlendSwitch
AND  CmdBlendSwitch
ST   SUP71.xBlendSwitchEn
ST   SUP72.xBlendSwitchEn
ST   SUP73.xBlendSwitchEn
ST   SUP74.xBlendSwitchEn
ST   SUP75.xBlendSwitchEn

LD   SupervisePos_X1
ST   SUP71.xSupervisePos
ST   SUP72.xSupervisePos
ST   SUP73.xSupervisePos
ST   SUP74.xSupervisePos
ST   SUP75.xSupervisePos

LD   OptEnabAutoPark
ANDN (
LD   IN_M700_M704
EQ   700
ANDN M700_BLEND
AND  %cn0.rc8.0
)
ST   SUP71.xEnabAutoUp
ST   SUP72.xEnabAutoUp
ST   SUP73.xEnabAutoUp
ST   SUP74.xEnabAutoUp
ST   SUP75.xEnabAutoUp

LD   IN_M700_M704
ST   SUP71.xM700_M704
ST   SUP72.xM700_M704
ST   SUP73.xM700_M704
ST   SUP74.xM700_M704
ST   SUP75.xM700_M704

LD   IN_M4_MODE
JMPCN NOG1000PRK
     LD   0
     ST   SUP71.xM700_M704
     ST   SUP72.xM700_M704
     ST   SUP73.xM700_M704
     ST   SUP74.xM700_M704
     ST   SUP75.xM700_M704
NOG1000PRK:

LD   OptEnabAutoPark
ST   SUP71.xEnabAutoDwn
ST   SUP72.xEnabAutoDwn
ST   SUP73.xEnabAutoDwn
ST   SUP74.xEnabAutoDwn
ST   SUP75.xEnabAutoDwn

LD   ParkingPositionUnload
ST   SUP71.xParkingPos
ST   SUP72.xParkingPos
ST   SUP73.xParkingPos
ST   SUP74.xParkingPos
ST   SUP75.xParkingPos

LD   UnloadSupQta
ST   SUP71.xUnSupQta
ST   SUP72.xUnSupQta
ST   SUP73.xUnSupQta
ST   SUP74.xUnSupQta
ST   SUP75.xUnSupQta

LD   20000
ST   SUP71.xAddFollPos
ST   SUP72.xAddFollPos
ST   SUP73.xAddFollPos
ST   SUP74.xAddFollPos
ST   SUP75.xAddFollPos

* [lv, lat, ulv, uhor]=[0,1,2,3]
LD   2
ST   SUP71.xBlendId
ST   SUP72.xBlendId
ST   SUP73.xBlendId
ST   SUP74.xBlendId
ST   SUP75.xBlendId

LD   %config_machine0.8
*ST   SUP71.xEnCyComSup
ST   SUP72.xEnCyComSup
ST   SUP73.xEnCyComSup
ST   SUP74.xEnCyComSup
ST   SUP75.xEnCyComSup
JMPCN _CYCOMOFT
LD   %ax61.ra24
*ST   SUP71.xCyComOft
ST   SUP72.xCyComOft
ST   SUP73.xCyComOft
ST   SUP74.xCyComOft
ST   SUP75.xCyComOft
_CYCOMOFT:

LD   %cn7.cc1.2
ST   SUP72.xEnBldFeed
LD   %cn7.cc1.3
ST   SUP73.xEnBldFeed
LD   %cn7.cc1.4
ST   SUP74.xEnBldFeed
LD   %cn7.cc1.5
ST   SUP75.xEnBldFeed

*******************************************************
*                      SUPPORT 1                      *
*******************************************************
LD   %cn8.cc1.1
JMPCN no_support_1

LD   MinPieceUnload
DIV  2
* Assuming 1/2 piece length falling down naturally
ABS
LT   TubeLengthInMach
ST   TubeReachSup_71

CAL  SUP71_ForceDwn(xIsoForce=iso_LsronCutting, xHoldMovSuperv=Hold_U_Z1Supp)

PATH  %ax71

LD   %ax36.ra4
LT   SafeDis_W_L1
ANDN iso_G520_Running
AND  %cn3.cc1.4                              * Exsisting V axis
JMPCN SECSUPERV
     LD   0
     ST   SUP71.xSupervisePos                * U posiz
SECSUPERV:

LD   OffsetUnSuppDwn_71
ST   SUP71.xSuperviseOft

LD   U_Posit_Z1_Down
ST   SUP71.xLimitSuppDwn

LD   %ax36.ra4
LT   SafeDis_W_L1
AND  iso_G520_Running
AND  %cn3.cc1.4                         * Exsisting V axis
OR   ParkUn72Sup_ISO
OR   ParkAllCmd
OR   SUP71_ForceDwn.yForceDwn
OR(
     LDN  TubeReachSup_71
     ANDN IN_M4_MODE
     *ANDN iso_G510_Running
     ANDN iso_G520_Running
     AND  %cn0.rc8.0
)
ST   SUP71.xParkCmd
ST   SUP71_xParkCmd

LD   TubeLengthInMach
LT   200000                             * 200mm tube length
AND  (
LD   TubeLengthInMach
GT   20
)
AND  AllowSecFTar
ST   SUP71.xEnSecFollow

LD   iso_G520_71_Unload
ST   SUP71.xG520VSup

CAL  SUP71

LD   SUP71.yReqGrant
ANDN ch8_in_ref
ST   usrReqGrantSup1

LD   SUP71.yHoldMovSupp
ANDN ch8_in_ref
ANDN ISO_SupUn_Init
ST   HoldZ1Supp

LD   SUP71.yHoldMovSuperv
ANDN ch8_in_ref
ST   Hold_U_Z1Supp

LD   SUP71.yAxInParkPos
ST   Z1Supp_71InParkPos

LD   SUP71.yCyComDwn
ST   yActivatedCyCom_71

LD   SUP71.yCyComOft
ST   CyComOftAx71

LDN  I_I_L1_Down
AND(
LD   U_Posit_Z1_Down
SUB  %ax71.ra4
ABS
LT   300              * 0.3mm
)
S    %PLCerr21.30

no_support_1:

LD   Pul_Reset
R    %PLCerr21.30

*******************************************************
*                      SUPPORT 2                      *
*******************************************************
LD   %cn8.cc1.2
JMPCN no_support_2

LD   U_Posit_Z2_Down
ADD  FlapWidth
ABS
LT   TubeLengthInMach
ST   TubeReachSup_72

CAL  SUP72_ForceDwn(xIsoForce=iso_LsronCutting, xHoldMovSuperv=Hold_U_Z2Supp)

PATH  %ax72

LD   OffsetUnSuppDwn_72
ST   SUP72.xSuperviseOft

LD   U_Posit_Z2_Down
ST   SUP72.xLimitSuppDwn

LD   ParkUn72Sup_ISO
OR   ParkAllCmd
OR   SUP72_ForceDwn.yForceDwn
OR(
     LDN  TubeReachSup_72
     ANDN IN_M4_MODE
     *ANDN iso_G510_Running
     ANDN iso_G520_Running
     AND  %cn0.rc8.0
)
ST   SUP72.xParkCmd
ST   SUP72_xParkCmd

LD   U_Posit_Z2_Down
ADD  FlapWidth
ABS
SUB  TubeLengthInMach
ABS
LT   100000                             * 100mm tube length
AND  AllowSecFTar
ST   SUP72.xEnSecFollow

LD   iso_G520_72_Unload
ST   SUP72.xG520VSup

LD   BLDFEED_72_85_Percent
ST   SUP72.xBldFeed

CAL  SUP72

LD   SUP72.yReqGrant
ANDN ch8_in_ref
ST   usrReqGrantSup2

LD   SUP72.yHoldMovSupp
ANDN ch8_in_ref
ANDN ISO_SupUn_Init
ST   HoldZ2Supp

LD   SUP72.yHoldMovSuperv
ANDN ch8_in_ref
ST   Hold_U_Z2Supp

LD   SUP72.yAxInParkPos
ST   Z2Supp_72InParkPos

LD   SUP72.yCyComDwn
ST   yActivatedCyCom_72

LD   SUP72.yCyComOft
ST   CyComOftAx72

no_support_2:

*******************************************************
*                      SUPPORT 3                     *
*******************************************************
LD   %cn8.cc1.3
JMPCN no_support_3

LD   U_Posit_Z3_Down
ADD  FlapWidth
ABS
LT   TubeLengthInMach
ST   TubeReachSup_73

CAL  SUP73_ForceDwn(xIsoForce=iso_LsronCutting, xHoldMovSuperv=Hold_U_Z3Supp)

PATH  %ax73

LD   OffsetUnSuppDwn_73
ST   SUP73.xSuperviseOft

LD   U_Posit_Z3_Down
ST   SUP73.xLimitSuppDwn

LD   ParkUn73Sup_ISO
OR   ParkAllCmd
OR   SUP73_ForceDwn.yForceDwn
OR(
     LDN  TubeReachSup_73
     ANDN IN_M4_MODE
     *ANDN iso_G510_Running
     ANDN iso_G520_Running
     AND  %cn0.rc8.0
)
*OR   Hor_Ax73_yVerForceDwn
ST   SUP73.xParkCmd
ST   SUP73_xParkCmd

LD   U_Posit_Z3_Down
ADD  FlapWidth
ABS
SUB  TubeLengthInMach
ABS
LT   100000                             * 100mm tube length
AND  AllowSecFTar
ST   SUP73.xEnSecFollow

LD   iso_G520_73_Unload
ST   SUP73.xG520VSup

LD   BLDFEED_73_86_Percent
ST   SUP73.xBldFeed

CAL  SUP73

LD   SUP73.yReqGrant
ANDN ch8_in_ref
ST   usrReqGrantSup3

LD   SUP73.yHoldMovSupp
ANDN ch8_in_ref
ANDN ISO_SupUn_Init
ST   HoldZ3Supp

LD   SUP73.yHoldMovSuperv
ANDN ch8_in_ref
ST   Hold_U_Z3Supp

LD   SUP73.yAxInParkPos
ST   Z3Supp_73InParkPos

LD   SUP73.yCyComDwn
ST   yActivatedCyCom_73

LD   SUP73.yCyComOft
ST   CyComOftAx73

no_support_3:

*******************************************************
*                      SUPPORT 4                     *
*******************************************************
LD   %cn8.cc1.4
JMPCN no_support_4

LD   U_Posit_Z4_Down
ADD  FlapWidth
ABS
LT   TubeLengthInMach
ST   TubeReachSup_74

CAL  SUP74_ForceDwn(xIsoForce=iso_LsronCutting, xHoldMovSuperv=Hold_U_Z4Supp)

PATH %ax74

LD   OffsetUnSuppDwn_74
ST   SUP74.xSuperviseOft

LD   U_Posit_Z4_Down
ST   SUP74.xLimitSuppDwn

LD   ParkUn74Sup_ISO
OR   ParkAllCmd
OR   SUP74_ForceDwn.yForceDwn
OR(
     LDN  TubeReachSup_74
     ANDN IN_M4_MODE
     *ANDN iso_G510_Running
     ANDN iso_G520_Running
     AND  %cn0.rc8.0
)
*OR   Hor_Ax74_yVerForceDwn
ST   SUP74.xParkCmd
ST   SUP74_xParkCmd

LD   U_Posit_Z4_Down
ADD  FlapWidth
ABS
SUB  TubeLengthInMach
ABS
LT   100000                             * 100mm tube length
AND  AllowSecFTar
ST   SUP74.xEnSecFollow

LD   iso_G520_74_Unload
ST   SUP74.xG520VSup

LD   BLDFEED_74_87_Percent
ST   SUP74.xBldFeed

CAL  SUP74

LD   SUP74.yReqGrant
ANDN ch8_in_ref
ST   usrReqGrantSup4

LD   SUP74.yHoldMovSupp
ANDN ch8_in_ref
ANDN ISO_SupUn_Init
ST   HoldZ4Supp

LD   SUP74.yHoldMovSuperv
ANDN ch8_in_ref
ANDN ISO_SupUn_Init
ST   Hold_U_Z4Supp

LD   SUP74.yAxInParkPos
ST   Z4Supp_74InParkPos

LD   SUP74.yCyComDwn
ST   yActivatedCyCom_74

LD   SUP74.yCyComOft
ST   CyComOftAx74

no_support_4:

*******************************************************
*                      SUPPORT 5                     *
*******************************************************
LD   %cn8.cc1.5
JMPCN no_support_5

LD   U_Posit_Z5_Down
ADD  FlapWidth
ABS
LT   TubeLengthInMach
ST   TubeReachSup_75

CAL  SUP75_ForceDwn(xIsoForce=iso_LsronCutting, xHoldMovSuperv=Hold_U_Z5Supp)

PATH  %ax75

LD   OffsetUnSuppDwn_75
ST   SUP75.xSuperviseOft

LD   U_Posit_Z5_Down                   * dwn limit for support
ST   SUP75.xLimitSuppDwn

LD   ParkUn75Sup_ISO
OR   ParkAllCmd
OR   SUP75_ForceDwn.yForceDwn
OR(
     LDN  TubeReachSup_75
     ANDN IN_M4_MODE
     *ANDN iso_G510_Running
     ANDN iso_G520_Running
     AND  %cn0.rc8.0
)
*OR   Hor_Ax75_yVerForceDwn
ST   SUP75.xParkCmd
ST   SUP75_xParkCmd

LD   U_Posit_Z5_Down
ADD  FlapWidth
ABS
SUB  TubeLengthInMach
ABS
LT   100000                             * 100mm tube length
AND  AllowSecFTar
ST   SUP75.xEnSecFollow

LD   iso_G520_75_Unload
ST   SUP75.xG520VSup

LD   BLDFEED_75_88_Percent
ST   SUP75.xBldFeed

CAL  SUP75

LD   SUP75.yReqGrant
ANDN ch8_in_ref
ST   usrReqGrantSup5

LD   SUP75.yHoldMovSupp
ANDN ch8_in_ref
ANDN ISO_SupUn_Init
ST   HoldZ5Supp

LD   SUP75.yHoldMovSuperv
ANDN ch8_in_ref
ANDN ISO_SupUn_Init
ST   Hold_U_Z5Supp

LD   SUP75.yAxInParkPos
ST   Z5Supp_75InParkPos

LD   SUP75.yCyComDwn
ST   yActivatedCyCom_75

LD   SUP75.yCyComOft
ST   CyComOftAx75

no_support_5:

********************************************************************************
* V Axis speed reduction in case of unloading axes in parking
* ---> Blendswitch (0 - 1000) maps to (100% - 10%) feedrate of V
********************************************************************************
LD    1000
ST    VSuppFeedReduction              * 1000 = 100%

* LD    EnWriteBlendSwitch
* AND(                                * Ensure V is on the right side
*       LD    %ax31.ra4
*       SUB   U_Posit_Z1_Down
* 	    LT    0
* )
* AND(                                * Ensure V is in parking zone
*       LD    %ax31.ra4
*       SUB   U_Posit_Z1_Down
* 	    ABS
* 	    LT    200000                  * Check inside the SuppFB, keep the value same
* )
* JMPCN AX72_IN_PARKING
*
*       LD    %ax71.ra4
*       SUB   ParkingPositionUnload
*       MULDIV(M=1000,D=ParkingPositionUnload)
*       ADD   1000
*       ST    VSuppFeedReduction
*
* AX72_IN_PARKING:

*//=============================================================================
*// Unloading Flaps On Each Support
*//=============================================================================
UNLOAD_FLAPS

*//=============================================================================
*// Unloading Cylinder Supports for Motor-Cylinder Combined Mode Usage
*//=============================================================================
LD     %PLCFLAGS.0
ST     M_HoldAx_V

LD     %config_machine0.8
JMPCN _CYCOMSEL
       UN_CYLINDER_SUPPORTS
_CYCOMSEL:

********************************************************************************
END_FUNCTION

(* ---- usrUnLoa.plc ---- *)
#funcdec "SPist.plc"

#include "usrMem.inc"
#include "Iol.inc"

VAR_IN_OUT
#include "usrIol.inc"
#include "mem.inc"
END_VAR

VAR
B1_B2_MOVE:        SINGLE_PISTON;
END_VAR

FUNCTION UNLOADER

*****LD   PRGRUN_CN0                     ** M0.0 cn0.rc8.0  Programma in corso
*****ST   B1_B2_MOVE.xAuto
*****
*****LD   Pul_Reset                      ** (gPlc0.3)Reset pushbutton
*****OR   Pul_Start                      ** (gPlc0.1)Start pushbutton
*****ST   B1_B2_MOVE.xReset
*****
*****LD   BtnGui_B1_B2_Open
*****ST   B1_B2_MOVE.xManualPlus
*****
*****LD   BtnGui_B1_B2_Close
*****ST   B1_B2_MOVE.xManualMinus
*****
*****LD   Fun_M336_Ch0
*****ST   B1_B2_MOVE.xAutoPlus
*****
*****LD   Fun_M337_Ch0
*****ST   B1_B2_MOVE.xAutoMinus
*****
*****LD   I_I_PRESSIONE_ARIA_IMPIANTO    ** **(Common for all pistons) %USR_M0
*****ST   B1_B2_MOVE.xAirPressure
*****
*****LD   I_I_B1_B2_OPEN
*****ST   B1_B2_MOVE.xSensorPlus
*****
*****LD   I_I_B1_B2_CLOSE
*****ST   B1_B2_MOVE.xSensorMinus
*****
*****LD   I_I_B1_B2_OPEN
*****ST   B1_B2_MOVE.xPlusAtInit
*****
*****LD   0
*****ST   B1_B2_MOVE.xSingleEffect
*****
*****LD   10000
*****ST   B1_B2_MOVE.xTimeOut
*****
*****LDN  I_I_EMERGENZA                  ** Machine OK (no EMERG.)
*****ST   B1_B2_MOVE.xEmerg
*****
*****CAL  B1_B2_MOVE
*****
*****LD   B1_B2_MOVE.yPistonPlus
*****ST   O_O_B1_B2_Open
*****
*****LD   B1_B2_MOVE.yAlarm
*****OR   I_I_B1_B2_ALARM
*****ST   %PLCerr21.8
*****
*****LD   B1_B2_MOVE.yPistonMinus
*****ST   O_O_B1_B2_Close

END_FUNCTION

(* ---- usrVshp.plc ---- *)
*************************************************************
*       V-shape management (based on centerings)            *
*************************************************************

#funcdec "SPist.plc"            ** SINGLE_PISTON definition

VAR
* Pneumatic loading supports
VShapeVertSup1:     SINGLE_PISTON;    ** V shape for loading tube
VShapeVertSup2:     SINGLE_PISTON;    ** V shape for loading tube
VShapeVertSup3:     SINGLE_PISTON;    ** V shape for loading tube
VShapeVertSup4:     SINGLE_PISTON;    ** V shape for loading tube

RT_ParkAllSupZBtn:          R_TRIG;
ParkAllSupZBtn:             BOOL;

#include "iof.inc"
#include "usrIof.inc"
END_VAR

VAR_IN_OUT
#include "usrIol.inc"
#include "mem.inc"
END_VAR

#include "Iol.inc"
#include "usrMem.inc"

FUNCTION V_SHAPE

CAL RT_ParkAllSupZBtn(CLK:=ParkAllLoadSuppCmd)
LD  RT_ParkAllSupZBtn.Q
S   ParkAllSupZBtn

LD  I_I_VshapeZ1_Dwn
AND I_I_VshapeZ2_Dwn
AND I_I_VshapeZ3_Dwn
AND I_I_VshapeZ4_Dwn
OR  Pul_Reset
R   ParkAllSupZBtn
*******************************************************
*         Staggered avoidance position                *
*******************************************************
LD   %ax30.ra0.0
JMPCN closeloop_active

    LD   %ax30.ra92
    ST   PosUMis

JMP no_loop
closeloop_active:

    LD   %ax30.ra4
    ST   PosUMis
no_loop:

************************************************************
* Auxiliary V shape 1
************************************************************
* {{{
    LD     PRGRUN_CN0                     ** M0.0 cn0.rc8.0  Programma in corso
    ST     VShapeVertSup1.xAuto

    LD     Pul_Reset                      ** (gPlc0.3) Reset pushbutton
    OR     Pul_Start                      ** (gPlc0.1) Start pushbutton
    ST     VShapeVertSup1.xReset

    LD     BtnGuiVshapeZ1_UP                 ** (%SUPPORTS_SYSTEM.GUI.2)
    OR     BtnGuiVshapeAllZ_UP               ** (%SUPPORTS_SYSTEM.GUI.0)
    ANDN   Force_Open_Center_1
    ST     VShapeVertSup1.xManualPlus

    LD     BtnGuiVshapeZ1_Dwn                ** (%SUPPORTS_SYSTEM.GUI.6)
    OR     BtnGuiVshapeAllZ_Dwn              ** (%SUPPORTS_SYSTEM.GUI.1)
    OR (
        LD  ParkAllSupZBtn
        AND I_I_Support_1_Dwn
    )
    OR (
        LD PosUMis
        SUB 200000                          ** value used inside SUPPORT function block (added to have syncronism)
        LT SUPPORT_1_Quota
    )
    ST     VShapeVertSup1.xManualMinus

    LD     Fun_M332_Ch0                     ** not used
    OR (
        LD     ch8_ValFunM                  ** not used
        EQ     332
    )
    OR     Fun_M445_Ch0                     ** Not used
    OR     Fun_M452_Ch0                      ** Open all centering
    ST     VShapeVertSup1.xAutoPlus

    LD     Fun_M333_Ch0                     ** not used
    OR(
        LD     ch8_ValFunM                  ** not used
        EQ     333
    )
    OR     Fun_M455_Ch0                     ** not used
    OR     Fun_M456_Ch0
    ST     VShapeVertSup1.xAutoMinus

    LD     I_I_PRESSIONE_ARIA_IMPIANTO    ** **(Common for all pistons) %USR_M0
    ST     VShapeVertSup1.xAirPressure

    LD     I_I_VshapeZ1_Up                   ** (%SUPPORTS_SYSTEM.IO0.8)
    ST     VShapeVertSup1.xSensorPlus

    LD     I_I_VshapeZ1_Dwn                  ** (%SUPPORTS_SYSTEM.IO0.12)
    ST     VShapeVertSup1.xSensorMinus

    LD     %PLCFLAGS.0                      ** Initial state UP
    ST     VShapeVertSup1.xPlusAtInit

    LD     %PLCFLAGS.0                      ** UP & DOWN managment
    ST     VShapeVertSup1.xSingleEffect

    LD     TimeOutPistonDown                ** (%SUPPORTS_SYSTEM.values21)
    ST     VShapeVertSup1.xTimeOut

    LDN    I_I_EMERGENZA                    ** Machine OK (no EMERG.)
    ST     VShapeVertSup1.xEmerg

    CAL    VShapeVertSup1

    LD     VShapeVertSup1.yPistonPlus
    ST     O_O_Ev_VShapeZ1_Up                ** (%SUPPORTS_SYSTEM.IO1.8)

    LD     VShapeVertSup1.yPistonMinus
    ST     O_O_Ev_VShapeZ1_Dwn               ** (%SUPPORTS_SYSTEM.IO1.12)

    LD     VShapeVertSup1.yAlarm
    ST     %PLCerr22.0                      ** Timeout: Loader V piston support 1
*}}}

************************************************************
* Auxiliary V shape 2
************************************************************
* {{{
    LD     PRGRUN_CN0                     ** M0.0 cn0.rc8.0  Programma in corso
    ST     VShapeVertSup2.xAuto

    LD     Pul_Reset                      ** (gPlc0.3) Reset pushbutton
    OR     Pul_Start                      ** (gPlc0.1) Start pushbutton
    ST     VShapeVertSup2.xReset

    LD     BtnGuiVshapeZ2_UP                 ** (%SUPPORTS_SYSTEM.GUI.3)
    OR     BtnGuiVshapeAllZ_UP               ** (%SUPPORTS_SYSTEM.GUI.0)
    ANDN   Force_Open_Center_2
    ST     VShapeVertSup2.xManualPlus

    LD     BtnGuiVshapeZ2_Dwn                ** (%SUPPORTS_SYSTEM.GUI.7)
    OR     BtnGuiVshapeAllZ_Dwn              ** (%SUPPORTS_SYSTEM.GUI.1)
    OR (
        LD  ParkAllSupZBtn
        AND I_I_Support_2_Dwn
    )
    OR (
        LD PosUMis
        SUB 200000                          ** value used inside SUPPORT function block (added to have syncronism)
        LT SUPPORT_2_Quota
    )
    ST     VShapeVertSup2.xManualMinus

    LD     Fun_M332_Ch0
    OR (
        LD     ch8_ValFunM
        EQ     332
    )
    OR     Fun_M445_Ch0
    OR     Fun_M452_Ch0                     ** Open all centering
    ST     VShapeVertSup2.xAutoPlus

    LD     Fun_M333_Ch0
    OR(
        LD     ch8_ValFunM
        EQ     333
    )
    OR     Fun_M455_Ch0
    OR     Fun_M457_Ch0
    ST     VShapeVertSup2.xAutoMinus

    LD     I_I_PRESSIONE_ARIA_IMPIANTO    ** **(Common for all pistons) %USR_M0
    ST     VShapeVertSup2.xAirPressure

    LD     I_I_VshapeZ2_Up                   ** (%SUPPORTS_SYSTEM.IO0.9)
    ST     VShapeVertSup2.xSensorPlus

    LD     I_I_VshapeZ2_Dwn                  ** (%SUPPORTS_SYSTEM.IO0.13)
    ST     VShapeVertSup2.xSensorMinus

    LD     %PLCFLAGS.0                      ** Initial state UP
    ST     VShapeVertSup2.xPlusAtInit

    LD     %PLCFLAGS.0                      ** UP & DOWN managment
    ST     VShapeVertSup2.xSingleEffect

    LD     TimeOutPistonDown                ** (%SUPPORTS_SYSTEM.values21)
    ST     VShapeVertSup2.xTimeOut

    LDN    I_I_EMERGENZA                    ** Machine OK (no EMERG.)
    ST     VShapeVertSup2.xEmerg

    CAL    VShapeVertSup2

    LD     VShapeVertSup2.yPistonPlus
    ST     O_O_Ev_VShapeZ2_Up                ** (%SUPPORTS_SYSTEM.IO1.9)

    LD     VShapeVertSup2.yPistonMinus
    ST     O_O_Ev_VShapeZ2_Dwn               ** (%SUPPORTS_SYSTEM.IO1.13)

    LD     VShapeVertSup2.yAlarm
    ST     %PLCerr22.1                      ** Timeout: Loader V piston support 2
*}}}

************************************************************
* Auxiliary V shape 3
************************************************************
* {{{
    LD     PRGRUN_CN0                     ** M0.0 cn0.rc8.0  Programma in corso
    ST     VShapeVertSup3.xAuto

    LD     Pul_Reset                      ** (gPlc0.3) Reset pushbutton
    OR     Pul_Start                      ** (gPlc0.1) Start pushbutton
    ST     VShapeVertSup3.xReset

    LD     BtnGuiVshapeZ3_UP                 ** (%SUPPORTS_SYSTEM.GUI.4)
    OR     BtnGuiVshapeAllZ_UP               ** (%SUPPORTS_SYSTEM.GUI.0)
    ANDN   Force_Open_Center_3
    ST     VShapeVertSup3.xManualPlus

    LD     BtnGuiVshapeZ3_Dwn                ** (%SUPPORTS_SYSTEM.GUI.8)
    OR     BtnGuiVshapeAllZ_Dwn              ** (%SUPPORTS_SYSTEM.GUI.1)
    OR (
        LD  ParkAllSupZBtn
        AND I_I_Support_3_Dwn
    )
    OR (
        LD PosUMis
        SUB 200000                          ** value used inside SUPPORT function block (added to have syncronism)
        LT SUPPORT_3_Quota
    )
    ST     VShapeVertSup3.xManualMinus

    LD     Fun_M332_Ch0
    OR (
        LD     ch8_ValFunM
        EQ     332
    )
    OR     Fun_M445_Ch0
    OR     Fun_M452_Ch0                     ** Open all centering
    ST     VShapeVertSup3.xAutoPlus

    LD     Fun_M333_Ch0
    OR(
        LD     ch8_ValFunM
        EQ     333
    )
    OR     Fun_M455_Ch0
    OR     Fun_M458_Ch0
    ST     VShapeVertSup3.xAutoMinus

    LD     I_I_PRESSIONE_ARIA_IMPIANTO    ** **(Common for all pistons) %USR_M0
    ST     VShapeVertSup3.xAirPressure

    LD     I_I_VshapeZ3_Up                   ** (%SUPPORTS_SYSTEM.IO0.10)
    ST     VShapeVertSup3.xSensorPlus

    LD     I_I_VshapeZ3_Dwn                  ** (%SUPPORTS_SYSTEM.IO0.14)
    ST     VShapeVertSup3.xSensorMinus

    LD     %PLCFLAGS.0                      ** Initial state UP
    ST     VShapeVertSup3.xPlusAtInit

    LD     %PLCFLAGS.0                      ** UP & DOWN managment
    ST     VShapeVertSup3.xSingleEffect

    LD     TimeOutPistonDown                ** (%SUPPORTS_SYSTEM.values21)
    ST     VShapeVertSup3.xTimeOut

    LDN    I_I_EMERGENZA                    ** Machine OK (no EMERG.)
    ST     VShapeVertSup3.xEmerg

    CAL    VShapeVertSup3

    LD     VShapeVertSup3.yPistonPlus
    ST     O_O_Ev_VShapeZ3_Up                ** (%SUPPORTS_SYSTEM.IO1.10)

    LD     VShapeVertSup3.yPistonMinus
    ST     O_O_Ev_VShapeZ3_Dwn               ** (%SUPPORTS_SYSTEM.IO1.14)

    LD     VShapeVertSup3.yAlarm
    ST     %PLCerr22.2                      ** Timeout: Loader V piston support 3
*}}}

************************************************************
* Auxiliary V shape 4
************************************************************
* {{{
    LD     PRGRUN_CN0                     ** M0.0 cn0.rc8.0  Programma in corso
    ST     VShapeVertSup4.xAuto

    LD     Pul_Reset                      ** (gPlc0.3) Reset pushbutton
    OR     Pul_Start                      ** (gPlc0.1) Start pushbutton
    ST     VShapeVertSup4.xReset

    LD     BtnGuiVshapeZ4_UP                 ** (%SUPPORTS_SYSTEM.GUI.5)
    OR     BtnGuiVshapeAllZ_UP               ** (%SUPPORTS_SYSTEM.GUI.0)
    ANDN   Force_Open_Center_4
    ST     VShapeVertSup4.xManualPlus

    LD     BtnGuiVshapeZ4_Dwn                ** (%SUPPORTS_SYSTEM.GUI.9)
    OR     BtnGuiVshapeAllZ_Dwn              ** (%SUPPORTS_SYSTEM.GUI.1)
    OR (
        LD  ParkAllSupZBtn
        AND I_I_Support_4_Dwn
    )
    OR (
        LD PosUMis
        SUB 200000                          ** value used inside SUPPORT function block (added to have syncronism)
        LT SUPPORT_4_Quota
    )
    ST     VShapeVertSup4.xManualMinus

    LD     Fun_M332_Ch0
    OR (
        LD     ch8_ValFunM
        EQ     332
    )
    OR     Fun_M445_Ch0
    OR     Fun_M452_Ch0                     ** Open all centering
    ST     VShapeVertSup4.xAutoPlus

    LD     Fun_M333_Ch0
    OR(
        LD     ch8_ValFunM
        EQ     333
    )
    OR     Fun_M455_Ch0
    OR     Fun_M459_Ch0
    ST     VShapeVertSup4.xAutoMinus

    LD     I_I_PRESSIONE_ARIA_IMPIANTO    ** **(Common for all pistons) %USR_M0
    ST     VShapeVertSup4.xAirPressure

    LD     I_I_VshapeZ4_Up                   ** (%SUPPORTS_SYSTEM.IO0.11)
    ST     VShapeVertSup4.xSensorPlus

    LD     I_I_VshapeZ4_Dwn                  ** (%SUPPORTS_SYSTEM.IO0.15)
    ST     VShapeVertSup4.xSensorMinus

    LD     %PLCFLAGS.0                      ** Initial state UP
    ST     VShapeVertSup4.xPlusAtInit

    LD     %PLCFLAGS.0                      ** UP & DOWN managment
    ST     VShapeVertSup4.xSingleEffect

    * LD     10000                            ** 10 sec
    LD     TimeOutPistonDown                ** (%SUPPORTS_SYSTEM.values21)
    ST     VShapeVertSup4.xTimeOut

    LDN    I_I_EMERGENZA                    ** Machine OK (no EMERG.)
    ST     VShapeVertSup4.xEmerg

    CAL    VShapeVertSup4

    LD     VShapeVertSup4.yPistonPlus
    ST     O_O_Ev_VShapeZ4_Up                ** (%SUPPORTS_SYSTEM.IO1.11)

    LD     VShapeVertSup4.yPistonMinus
    ST     O_O_Ev_VShapeZ4_Dwn               ** (%SUPPORTS_SYSTEM.IO1.15)

    * LD     VShapeVertSup4.yAlarm
    * AND    SUPPORT_4.xEnable                ** Provisional
    * ST     %PLCerr22.3                      ** Timeout: Loader V piston support 4
*}}}

LD   I_I_VshapeZ1_Dwn
AND  I_I_VshapeZ2_Dwn
AND  I_I_VshapeZ3_Dwn
AND  I_I_VshapeZ4_Dwn
ST   All_Vshape_DWN

END_FUNCTION

(* ---- VRTCTEST.PLC ---- *)
#include "iol.inc"

VAR

RTRIG_PROGRUN: R_TRIG;

loadconfig:    DWORD;
calcBeam:      DWORD;

END_VAR

FUNCTION VRTC_TEST
********************************************************************************

* FOX=0,FOY=0,FOZ=0) ORIGINE PIANO
* FRX=0,FRY=0,FRZ=0 MILIONESIMI DI GRADO ESPRIMO ROTAZIONE SU UN ASSE

CAL  RTRIG_PROGRUN (CLK:=PRGRUN_CN0)

* Test Vrtc

LD   RTRIG_PROGRUN.Q
JMPCN  no_load_wjs1

LD   0               * N/C
WJS_LOAD (INS=3,CH=3,TWI=1,THD=1,CED=1,SVL=0,CHX=0,CHY=1,CHZ=2,FRX=%M161,FRY=0,FRZ=0,FOX=0,FOY=0,FOZ=0)
ST   loadconfig      * 0 = OK
no_load_wjs1:

LD   loadconfig
NE   0
JMPC errorAngle

LD      0               * N/C
WJS_BEAM_CALC (INS=3,SVL=0)
ST      calcBeam            * 0 = OK

LD      calcBeam
NE      0
JMPC    errorAngle

*  Tilt angle

LD      0               * N/C
WJS_GETZ_FTCP (INS=3)   * DISTANZA DAL PIANO (ORTOGONALE ) per simulazione capacitivo e monitoraggio
ST   DistZPianoSimul

LD      0               * N/C
WJS_GETX_M (INS=3)             * coordinata X/Y/Z di intersezione col piano. monitor deviazione traiettoria
ST   x_TCPDeviaz

LD      0               * N/C
WJS_GETY_M(INS=3)              * coordinata X/Y/Z di intersezione col piano. monitor deviazione traiettoria
ST   y_TCPDeviaz

LD      0               * N/C
WJS_GETZ_M(INS=3)             * coordinata X/Y/Z di intersezione col piano.  monitor altezza piano nel punto di intersezione
ST   Z_TCPDeviaz

LD      0               * N/C
WJS_DIST_T(INS=3)              * Ritorna la distanza col segno del TCP dal punto di intersezione col piano. monitor stand off istantaneo
ST   StandOff_Calc
*****
* creare nuova istanza wjs con le quote calcolate ch0

LD   RTRIG_PROGRUN.Q
JMPCN no_load_wjs

LD   0               * N/C
WJS_LOAD (INS=6,CH=3,TWI=1,THD=1,CED=1,SVL=0,CHX=16#40000000,CHY=16#40000001,CHZ=16#40000002,FRX=0,FRY=0,FRZ=0,FOX=0,FOY=0,FOZ=0)
ST   loadconfig      * 0 = OK

no_load_wjs:

LD   loadconfig
NE   0
JMPC errorAngle

LD      0               * N/C
WJS_BEAM_CALC (INS=6,SVL=0)
ST      calcBeam            * 0 = OK

LD      calcBeam
NE      0
JMPC    errorAngle

LD      0               * N/C
WJS_GETX_TCP(INS=6)            * Ritorna la coordinata X/Y/Z del TCP.
ST   X_TCP

LD      0               * N/C
WJS_GETY_TCP(INS=6)            * Ritorna la coordinata X/Y/Z del TCP.
ST   Y_TCP

* ra54 cn0 Quota asse riferita al TCP. Attenzione alla rotazione origini

JMP noerror
errorAngle:

LD   1
S    %PLCerr8.31
noerror:

LD   Pul_Reset
R    %PLCerr8.31ù

END_FUNCTION

(* ---- AntiAtoS.plc ---- *)
*****************************************************************************************************
* Used for One Axes Anti-collision with Support(Obstercal) Control(Duo)
*
* The function is based on AO_DYN_TARGET 92
*
* #funcdec "AntiAtoS.plc"
* ANTIAXIS:              ANTI_AXIS_SUPPORT;
*
* CAL ANTIAXIS(xEnable:=,xAx_Num:=,xObs_Qta:=,xDisSafe:=,xReset:=)
* LD  ANTIAXIS.yHoldMov *---> Pul_Stop, .xJogMinus , .xJogPlus, xHoldMoving
*****************************************************************************************************

FUNCTION_BLOCK  ANTI_AXIS_SUPPORT
*****************************************************************************************************
* The Function Block to prevent two axes collide
*****************************************************************************************************

VAR_INPUT
xEnable:           BOOL;          * Enable
xReset:            BOOL;          * To Reset the Anticolision Alarm
xAx_Num:           DWORD;         * Axis ID
xObs_Qta:          DWORD;         * [um]The Obstercal Abs Quota(one side, if two side using two FB)
xDisSafe:          DWORD;         * [um]Safe Distance Between Two Heads(Exact Speed 0)
xColiDir:          DWORD;         * Colisiion direction 0 = BOTH, 1 = POS, 2 = NEG
END_VAR

VAR_OUTPUT
yHoldMov:          BOOL;          * Hold Ax and STOP at calculated distance
END_VAR

VAR
ZeroSpeed:         BOOL;
Ax_Plus:           BOOL;
Ax_Minus:          BOOL;
ColisionDirection: BOOL;
Ax_Ferma:          BOOL;
HoldPos:           BOOL;
HoldNeg:           BOOL;
HoldMov:           BOOL;
OnlyMovPos:        BOOL;
OnlyMovNeg:        BOOL;
BothDir:           BOOL;
Ax_dcc:           DWORD;
Ax_speed:         DWORD;
Ax_Quota:         DWORD;
Ax_AvaQta:        DWORD;
END_VAR

*****************************************************************************************************
PATH     %ax[xAx_Num]

LD       %ra24
ST       Ax_Quota               *um

LD       %pa2
ST       Ax_dcc                 *mm/s2

LD       %ra3.2                 * ra3.2  Direzione moto asse avanti
OR       %ra0.8                 * ra0.8 Comando avanti
AND      %ra3.13                * ra3.13  Ordine di moto
AND      %cn0.rc8.0
OR(
LD       %ra0.8                 * ra0.8 Comando avanti
ANDN     %cn0.rc8.0
)
ST       Ax_Plus

LDN      %ra3.2                 * ra3.2  Direzione moto asse avanti
OR       %ra0.9                 * ra0.9 Comando indietro
AND      %ra3.13                * ra3.13  Ordine di moto
AND      %cn0.rc8.0
OR(
LD       %ra0.9                 * ra0.9 Comando indietro
ANDN     %cn0.rc8.0
)
ST       Ax_Minus

LD       %ra3.0
ST       Ax_Ferma

LD       %ra92
ST       Ax_AvaQta              *um

LD       xReset
OR       %PLCFLAGS.8
JMPCN    INITOUTPUT
LD       0
ST       HoldMov
ST       yHoldMov
INITOUTPUT:

LD       xColiDir
EQ       0
ST       BothDir

LD       xColiDir
EQ       1
ST       OnlyMovPos

LD       xColiDir
EQ       2
ST       OnlyMovNeg

*****************************************************************************************************
* Only when moving towards each other activates it
*****************************************************************************************************
LD       xObs_Qta
GT       Ax_AvaQta             *Ax_Quota
AND      Ax_Plus
ANDN     OnlyMovNeg
OR(
LD       xObs_Qta
LT       Ax_AvaQta             *Ax_Quota
AND      Ax_Minus
ANDN     OnlyMovPos
)
ST       ColisionDirection

LD       ColisionDirection
AND      xEnable
AND(
LD       xDisSafe
GT       0
)
ANDN     yHoldMov
JMPCN    ANTICOLISIONCAL

*****************************************************************************************************
* Calculate the Position to apply hold axis and stop
*****************************************************************************************************
LD       Ax_AvaQta
SUB      xDisSafe
LT       xObs_Qta
AND      Ax_Minus
ST       HoldNeg

LD       Ax_AvaQta
ADD      xDisSafe
GT       xObs_Qta
AND      Ax_Plus
ST       HoldPos

LD       HoldNeg
OR       HoldPos
ST       HoldMov

ANTICOLISIONCAL:

*****************************************************************************************************
* FB Outputs Section
*****************************************************************************************************
LD       HoldMov
AND      ColisionDirection
ANDN     xReset
S        yHoldMov

LD       xReset
OR(
LD       HoldPos
AND      Ax_Minus
ANDN     %cn0.rc8.0
)
OR(
LD       HoldNeg
AND      Ax_Plus
ANDN     %cn0.rc8.0
)
ORN      xEnable
R        HoldMov
R        yHoldMov

*****************************************************************************************************
END_FUNCTION_BLOCK

(* ---- Antictrl.plc ---- *)
*************************************************************************************
* Used for 2 Axes Anti-collision Control(Duo)
*
* The function is based on AO_DYN_TARGET 92
*
* CAL ANTIAXIS(xAx1_Fst:=,xReset:=,xAx1_Num:=,xAx2_Num:=,xDisSafe:=)
* LD  ANTIAXIS.yHoldMov ---> Pul_Stop, .xJogMinus , .xJogPlus, xHoldMoving
* LD  ANTIAXIS.yDisSafeCal
*************************************************************************************

FUNCTION_BLOCK  ANTI_AXIS
*************************************************************************************
* The Function Block to prevent two axes collide
*************************************************************************************

VAR_INPUT
xAx1_Fst:          BOOL;          * TRUE when Ax1 is more near to the origin
xReset:            BOOL;          * To Reset the Anticolision Alarm
xAx1_Num:          DWORD;         * Axis 1 ID
xAx2_Num:          DWORD;         * Axis 2 ID
xDisSafe:          DWORD;         * [um]Safe Distance Between Two Heads(Exact Speed 0)
END_VAR

VAR_OUTPUT
yHoldMov:          BOOL;          * Hold Ax and STOP at calculated distance
yDisSafeCal:       DWORD;         * [um]The distance start to stop(to show gui or debug)
END_VAR

VAR
PowerOn:           BOOL;
DangerZone:        BOOL;
ZeroSpeed:         BOOL;
CaseToEach1:       BOOL;
CaseToEach2:       BOOL;
Ax1_Go_Cn:          BOOL;
Ax2_Go_Cn:          BOOL;
Ax1_Plus:          BOOL;
Ax1_Minus:         BOOL;
Ax2_Plus:          BOOL;
Ax2_Minus:         BOOL;
HoldMov:           BOOL;
InPosLimit:        BOOL;
JogSafeDirection:  BOOL;
DisTDelay:         DWORD;
DisSafeCal:        DWORD;
DeltaDis1:         DWORD;
DeltaDis2:         DWORD;
Ax1_dcc:           DWORD;
Ax2_dcc:           DWORD;
Ax1_speed:         DWORD;
Ax2_speed:         DWORD;
Ax1_Quota:         DWORD;
Ax2_Quota:         DWORD;
Ax1_AvaQta:        DWORD;
Ax2_AvaQta:        DWORD;
Ax1_MinQta:        DWORD;
Ax2_MinQta:        DWORD;
Ax1_MaxQta:        DWORD;
Ax2_MaxQta:        DWORD;
END_VAR

*************************************************************************************
PATH     %ax[xAx1_Num]

LD       %ra3.10
ST       PowerOn

LD       %ra4                    *
ST       Ax1_Quota

LD       %ra3.13               * ra3.13  Ordine di moto
*AND      %ra3.0
ST       Ax1_Go_Cn

LD       %ra5
DIV      1000
ST       Ax1_speed             *um/s

LD       %pa2
ST       Ax1_dcc               *mm/s2

LD       %ra3.2                 * ra3.2  Direzione moto asse avanti
OR       %ra0.8                 * ra0.8 Comando avanti
AND      %ra3.13                * ra3.13  Ordine di moto
AND      %cn0.rc8.0
OR(
LD       %ra0.8                 * ra0.8 Comando avanti
AND      %ra3.13                * ra3.13  Ordine di moto
ANDN     %cn0.rc8.0
)
ST       Ax1_Plus

LDN      %ra3.2                 * ra3.2  Direzione moto asse avanti
OR       %ra0.9                 * ra0.9 Comando indietro
AND      %ra3.13                * ra3.13  Ordine di moto
AND      %cn0.rc8.0
OR(
LD       %ra0.9                 * ra0.9 Comando indietro
AND      %ra3.13                * ra3.13  Ordine di moto
ANDN     %cn0.rc8.0
)
ST       Ax1_Minus

LD       %pa21
ST       Ax1_MinQta

LD       %pa22
ST       Ax1_MaxQta

LD       %ra92
ST       Ax1_AvaQta

PATH     %ax[xAx2_Num]

LD       %ra4
ST       Ax2_Quota

LD       %ra3.13               * ra3.13  Ordine di moto
*AND      %ra3.0
ST       Ax2_Go_Cn

LD       %ra5                    *um/s
DIV      1000
ST       Ax2_speed               *mm/s

LD       %pa2
ST       Ax2_dcc                 *mm/s2

LD       %ra3.2                 * ra3.2  Direzione moto asse avanti
OR       %ra0.8                 * ra0.8 Comando avanti
AND      %ra3.13                * ra3.13  Ordine di moto
AND      %cn0.rc8.0
OR(
LD       %ra0.8                 * ra0.8 Comando avanti
AND      %ra3.13                * ra3.13  Ordine di moto
ANDN     %cn0.rc8.0
)
ST       Ax2_Plus

LDN      %ra3.2                 * ra3.2  Direzione moto asse avanti
OR       %ra0.9                 * ra0.9 Comando indietro
AND      %ra3.13                * ra3.13  Ordine di moto
AND      %cn0.rc8.0
OR(
LD       %ra0.9                 * ra0.9 Comando indietro
AND      %ra3.13                * ra3.13  Ordine di moto
ANDN     %cn0.rc8.0
)
ST       Ax2_Minus

LD       %pa21
ST       Ax2_MinQta

LD       %pa22
ST       Ax2_MaxQta

LD       %ra92
ST       Ax2_AvaQta

LD       Ax1_Quota
SUB      Ax2_Quota
ABS
LT       xDisSafe
ST       DangerZone

LD       xReset
ANDN     DangerZone
OR       %PLCFLAGS.8
ORN      PowerOn
JMPCN    INITOUTPUT
LD       xDisSafe
ST       DisSafeCal
ST       yDisSafeCal
LD       %PLCFLAGS.0
ST       HoldMov
ST       yHoldMov
INITOUTPUT:

*************************************************************************************
* Only when the two axis moving towards each other activates it
*************************************************************************************
LD       Ax1_speed
EQ       0
AND(
LD       Ax2_speed
EQ       0
)
ST       ZeroSpeed

LD       Ax1_speed
GE       0
AND(
LD       Ax2_speed
LE       0
)
AND      xAx1_Fst
ST       CaseToEach1

LD       Ax1_speed
LE       0
AND(
LD       Ax2_speed
GE       0
)
ANDN     xAx1_Fst
ST       CaseToEach2

LD       CaseToEach1
OR       CaseToEach2
*ANDN     ZeroSpeed
OR(
LD       Ax1_Minus
AND      Ax2_Minus
)
OR(
LD       Ax1_Plus
AND      Ax2_Plus
)
AND(
LD       xDisSafe
GT       0
)
ANDN     yHoldMov
JMPCN    ANTICOLISIONCAL

*************************************************************************************
* Calculate the Position to apply hold axis and stop
* Only Consider the case of consistent speed(Jog Mode)
*************************************************************************************
LD       Ax1_AvaQta
SUB      Ax2_AvaQta
ABS
LE       DisSafeCal
OR       DangerZone
AND      PowerOn
ST       HoldMov

ANTICOLISIONCAL:

LD       Ax1_Minus
OR       Ax2_Plus
AND      xAx1_Fst
OR(
LD       Ax2_Minus
OR       Ax1_Plus
ANDN     xAx1_Fst
)
ANDN(
LD       Ax1_Minus
AND      Ax2_Minus
)
ANDN(
LD       Ax1_Plus
AND      Ax2_Plus
)
ST       JogSafeDirection

*************************************************************************************
* FB Outputs Section
*************************************************************************************
LD       DisSafeCal
ST       yDisSafeCal

LD       HoldMov
ANDN     JogSafeDirection
S        yHoldMov

LD       JogSafeDirection
ANDN(
LD       Ax1_Go_Cn
AND      Ax2_Go_Cn
)
R        HoldMov
R        yHoldMov

*************************************************************************************
END_FUNCTION_BLOCK
